           END_IF;
           //END_IF of IF #si_WDOG_RETRY < #si_WDOG_RETRY_NO 

         ELSE
           ;
           //keine Bedeutung 
         END_IF;
         //END_IF of IF #BUSY 

       END_IF;
       //END_IF of IF (NOT #BUSY AND #START AND NOT #sb_START_OLD) OR (#BUSY AND #sb_SEND)

     ELSE
       ;
       //Konfigurationsfehler: keine weitere Bearbeitung 

       #sb_CFG_ERR_1 := TRUE;

       //Auftrag ist nicht aktiv 

       #sb_BUSY := FALSE;

       //Auftrag fertig ruecksetzen 

       #sb_DONE := FALSE;
     END_IF;
     //END_IF of IF #LADDR <> 16#0000 

     //Flankenauswertung Startimpuls 

     #sb_START_OLD := #START;

     //CFG_ERR ausgeben 

     #CFG_ERR := #sb_CFG_ERR_1;

     //DB_ERR ausgeben 

     #DB_ERR := #sb_DB_ERR;

     // Initialisierung von Ausg㭧en
     #BUSY := #sb_BUSY;
     #DONE := #sb_DONE;
     #REQ_ERR := #sb_REQ_ERR;
END_FUNCTION_BLOCK

// ===== library: MasterCopy "DEV_FLT4" =====

FUNCTION_BLOCK "DEV_FLT4"   // FB39, SCL
TITLE = DEV_FLT4
{ S7_Optimized_Access := 'TRUE' }
AUTHOR : DRVDPS7
FAMILY : DRIVES
NAME : DEV_FLT4
VERSION : 5.0
// Read out fault buffer of a SINAMICS (CPU 1200)
   VAR_INPUT
      LADDR : Hw_Io;   // Logic base address of slot
      DS_NO : Word := 0;   // Number of data record
      AXIS : Byte;   // Axis addressing for multi-axis drives / Axis addressing
      START : Bool;   // Accept start impulse for request
   END_VAR
   VAR_OUTPUT
      BUSY : Bool;   // Request busy
      DONE : Bool := 1;   // Request completed without error
      REQ_ERR : Bool;   // Request completed with error
      WDOG_ERR : Bool;   // Watchdog error, no plausible response data exist
      SFB_ERR : Bool;   // SFB 53 WRREC / SFB 52 RDREC signals error
      CFG_ERR : Bool;   // Slave incorrectly configured or not at all
      ERR_NO1 : Word;   // Number fault 1 of fault event
      ERR_VAL1 : DWord;   // Fault value for fault number of fault 1
      ERR_NO2 : Word;   // Number fault 2 of fault event
      ERR_VAL2 : DWord;   // Fault value for fault number of fault 2
      ERR_NO3 : Word;   // Number fault 3 of fault event
      ERR_VAL3 : DWord;   // Fault value for fault number of fault 3
      ERR_NO4 : Word;   // Number fault 4 of fault event
      ERR_VAL4 : DWord;   // Fault value for fault number of fault 4
      ERR_NO5 : Word;   // Number fault 5 of fault event
      ERR_VAL5 : DWord;   // Fault value for fault number of fault 5
      ERR_NO6 : Word;   // Number fault 6 of fault event
      ERR_VAL6 : DWord;   // Fault value for fault number of fault 6
      ERR_NO7 : Word;   // Number fault 7 of fault event
      ERR_VAL7 : DWord;   // Fault value for fault number of fault 7
      ERR_NO8 : Word;   // Number fault 8 of fault event
      ERR_VAL8 : DWord;   // Fault value for fault number of fault 8 statische Variablen
   END_VAR
   VAR
      SFB53_RET_VAL : Int;   // Return value of SFB 53 WRREC
      SFB52_RET_VAL : Int;   // Return value of SFB 52 RDREC
      WDOG_RETRY_NO : Byte := BYTE#16#05;   // Number of request retries, when no plausible response data exists
      NODATA_RETRY_NO : Byte := BYTE#16#05;   // Number of request retries, when no response data exist
      NODATA_CYCLE_NO : Int := 2500;   // Number of cycles when no response data exist, before request retry
      sx_SEND_FA : Struct   // send buffer
         sy_AR : Byte;   // Auftragsreferenz
         sy_AKE : Byte := BYTE#16#01;   // Auftragskennung: 16#01 (Parameter anfordern )
         sy_A_NO : Byte := BYTE#16#00;   // Achsnummer
         sy_ANZ_PARA : Byte := BYTE#16#02;   // Anzahl Parameter: 16#02
         sy_ATTRIB1 : Byte := BYTE#16#10;   // Attribut: 16#10 (Wert)
         sy_ANZ_ELEM1 : Byte := BYTE#16#08;   // Anzahl Arrayelemente: 16#08
         si_PARA_NO1 : Int := 947;   // Parameternummer: 947 (Stoernummer)
         si_SUB_IND1 : Int := 0;   // Subindex: 0 (adressiert erstes Arrayelement auf das zugegriffen wird)
         sy_ATTRIB2 : Byte := BYTE#16#10;   // Attribut: 16#10 (Wert)
         sy_ANZ_ELEM2 : Byte := BYTE#16#08;   // Anzahl Arrayelemente: 16#08
         si_PARA_NO2 : Int := 949;   // Parameternummer: 949 (Stoerwert)
         si_SUB_IND2 : Int := 0;   // Subindex: 0 (adressiert erstes Arrayelement auf das zugegriffen wird)
      END_STRUCT;
      sx_RECV_FA : Struct   // receive buffer
         sy_AR : Byte;   // gespiegelte Auftragsreferenze
         sy_AKE : Byte;   // Antwortkennung
         sy_A_NO : Byte;   // Achsnummer
         sy_ANZ_PARA : Byte;   // Anzahl Parameter
         sy_FORMAT1 : Byte;   // Format
         sy_ANZ_VAL1 : Byte;   // Anzahl Werte
         sw_FAULT_NO1 : Word;   // Stoernummer 1
         sw_FAULT_NO2 : Word;   // Stoernummer 2
         sw_FAULT_NO3 : Word;   // Stoernummer 3
         sw_FAULT_NO4 : Word;   // Stoernummer 4
         sw_FAULT_NO5 : Word;   // Stoernummer 5
         sw_FAULT_NO6 : Word;   // Stoernummer 6
         sw_FAULT_NO7 : Word;   // Stoernummer 7
         sw_FAULT_NO8 : Word;   // Stoernummer 8
         sy_FORMAT2 : Byte;   // Format
         sy_ANZ_VAL2 : Byte;   // Anzahl Werte
         sd_FAULT_VAL1 : DWord;   // Stoerwert 1
         sd_FAULT_VAL2 : DWord;   // Stoerwert 2
         sd_FAULT_VAL3 : DWord;   // Stoerwert 3
         sd_FAULT_VAL4 : DWord;   // Stoerwert 4
         sd_FAULT_VAL5 : DWord;   // Stoerwert 5
         sd_FAULT_VAL6 : DWord;   // Stoerwert 6
         sd_FAULT_VAL7 : DWord;   // Stoerwert 7
         sd_FAULT_VAL8 : DWord;   // Stoerwert 8
      END_STRUCT;
      WDOG_RETRY : Byte;   // Counter for request retry for Watchdog monitoring
      NODATA_RETRY : Byte;   // Counter for request retry, if no response data exist
      NODATA_CYCLE : Int;   // Cycle counter, if no reponse data exist
      SEND_AC : Bool;   // Transmission active or request repetition for acyclic Communication
      START_AC : Bool;   // Start pulse for acyclic Communication
      BUSY_AC : Bool;   // Request busy for acyclic Communication
      READY_AC : Bool;   // Request completed without error for Acyclic communication
      SEND : Bool;   // send next request
      sb_DONE_AC : Bool;   // Stoerspeicher auslesen beendet
      sb_BUSY : Bool;   // Request busy
      sb_REQ_ERR : Bool;   // Request completed with error
      sb_WDOG_ERR : Bool;   // Watchdog error, no plausible response data exist
      sb_SFB_ERR : Bool;   // SFB 53 WRREC / SFB 52 RDREC signals error
      sb_CFG_ERR : Bool;   // Slave incorrectly configured or not at all
      si_AUF_REF : Int;   // Auftragsreferenz
      HM_RET_VAL : Int;   // Return value of SFB
      sb_START_OLD : Bool := 0;   // Start flag
      WRREC_1 : WRREC;   // Multiinstance of WRREC (SFB53)
      RDREC_1 : RDREC;   // Multiinstance of RDREC (SFB52) temporaere Variablen
   END_VAR
   VAR_TEMP
      pd_STATUS : DWord;   // STATUS der SFB's
      w_p_no : Word;   // Zwischenspeicher fuer Parameter-Nummer
      i_index : Int;   // Hilfsmerker fuer Index
      pi_LEN_RDREC : UInt;   // Tatsaechliche Laenge der empfangenen Daten
      pi_SFB_INDEX : Int;   // Index bei SFB52/53 Aufruf
      y_page_sel : Byte;   // Hilfsmerker PARA PAGE SELECT Funktion
      b_pind : Bool;   // Hilfsmerker Parameter-Index Sendefach Empfangsfach gleich
      b_busy : Bool;   // SFB 53 WRREC / SFB 52 RDREC sind beschaeftigt
      pb_DONE_WRREC : Bool;   // WRREC fertig
      pb_DONE_RDREC : Bool;   // RDREC fertig
      pb_ERR_WRREC : Bool;   // WRREC Fehler
      pb_ERR_RDREC : Bool;   // RDREC Fehler
   END_VAR
BEGIN
     //=============================================================================
     //SIEMENS AG
     //(c)Copyright 2017 All Rights Reserved
     //-----------------------------------------------------------------------------
     // Library: DriveLib
     // Tested with: S7-1200 CPU 1212C DC/DC/DC V4.1
     // Engineering: TIA Portal V14
     // Restrictions: -
     // Requirements: S7-1200
     // Functionality: The block reads out the last fault stored in the fault memory of the drive.
     //=============================================================================

     //Stoerungen lesen: Auftrag anstossen 

     //Startimpuls vorhanden und kein Auftrag aktiv 

     IF #START AND NOT #sb_BUSY AND NOT #sb_START_OLD
     THEN
       //Fehler / Ausgaenge abloeschen 

       #DONE := FALSE;
       #sb_REQ_ERR := FALSE;
       #sb_SFB_ERR := FALSE;
       #sb_CFG_ERR := FALSE;

       #sb_DONE_AC := FALSE;
     END_IF;
     //END_IF of IF #START AND NOT #BUSY AND NOT #sb_START_OLD

     //Startimpuls vorhanden oder Anforderung naechsten Auftrag zu senden vorhanden 

     IF #START AND NOT #sb_START_OLD OR #SEND
     THEN
       IF (#si_AUF_REF > 254) OR (#si_AUF_REF <= 0)
       THEN
         #si_AUF_REF := 1;
       ELSE
         ;
         #si_AUF_REF := #si_AUF_REF + 1;
       END_IF;
       //END_IF of IF (#si_AUF_REF > 254) OR (#si_AUF_REF <= 0)
       //Startimpuls fuer azyklischen Kommunikation setzen 

       #START_AC := TRUE;

       //Stoerungen auslesen ist aktiv 

       #sb_BUSY := TRUE;

       //Anforderung naechsten Auftrag senden ruecksetzen 

       #SEND := FALSE;
     ELSE
       ;
       //Startimpuls fuer azyklischen Kommunikation ruecksetzen 

       #START_AC := FALSE;
     END_IF;
     //END_IF of IF #START AND NOT #sb_START_OLD OR #SEND

     //Flankenauswertung Startimpuls 

     #sb_START_OLD := #START;

     //Ãœberpruefung, welcher Datensatz verwendet werden soll 

     #pi_SFB_INDEX := WORD_TO_INT(#DS_NO);

     IF #pi_SFB_INDEX = 0
     THEN
       #pi_SFB_INDEX := 47;
     ELSE
       ;
       ;    // not used
     END_IF;
     //END_IF of IF #pi_SFB_INDEX = 0

     //PDAT_AC2: Azyklische Kommunikation 

     //Hilfsmerker ruecksetzen 

     //Hilfsmerker ruecksetzen 

     #b_pind := FALSE;
     #y_page_sel := 16#00;
     #w_p_no := 16#0000;
     #i_index := 0;

     //Konfigurationsdaten pruefen: Slot = PKW-Slot und Logische Basisadresse <> 0 

     IF (#LADDR <> 16#0000)
     THEN
       //Konfiguration o.k. 

       #sb_CFG_ERR := FALSE;

       //Auftrag laeuft 

       IF #BUSY_AC
       THEN
         //Anzahl Zyklen, wenn keine Antwortdaten vorhanden, noch nicht abgelaufen  

         IF #NODATA_CYCLE < #NODATA_CYCLE_NO
         THEN
           //Anzahl Zyklen erhoehen 

           #NODATA_CYCLE := #NODATA_CYCLE + 1;
         ELSE
           ;
           //Fehler vorhanden: Return-Wert der SFBs < 0 

           IF #HM_RET_VAL < 0
           THEN
             //Keine Antwortdaten vorhanden oder temporaerer Fehler? 

             //Anzahl Auftragswiederholungen, wenn keine Antwortdaten vorhanden, noch nicht abgelaufen 

             IF #NODATA_RETRY < #NODATA_RETRY_NO
             THEN
               //Anzahl Auftragswiederholungen, wenn keine Antwortdaten vorhanden, erhoehen 

               #NODATA_RETRY := #NODATA_RETRY + 1;

               //Anzahl Zyklen initialisieren 

               #NODATA_CYCLE := 0;
             ELSE
               ;
               //SFB-Fehler 

               #sb_SFB_ERR := TRUE;

               IF #SEND_AC
               THEN
                 //Datensatz schreiben:                                                   
                 //Keine Antwortdaten vorhanden oder temporaerer Fehler, RET_VAL uebergeben 

                 #SFB53_RET_VAL := #HM_RET_VAL;
               ELSE
                 ;
                 //Datensatz lesen:                                                       
                 //Keine Antwortdaten vorhanden oder temporaerer Fehler, RET_VAL uebergeben 

                 #SFB52_RET_VAL := #HM_RET_VAL;
               END_IF;
               //END_IF of IF 
               //Auftragswiederholung ruecksetzen 

               #SEND_AC := FALSE;

               //Auftrag nicht aktiv 

               #BUSY_AC := FALSE;
             END_IF;
             //END_IF of IF #NODATA_RETRY < #NODATA_RETRY_NO
           END_IF;
           //END_IF of IF #HM_RET_VAL < 0
         END_IF;
         //END_IF of IF #NODATA_CYCLE < #NODATA_CYCLE_NO
       ELSE
         ;
         //Anzahl Zyklen und Anzahl Auftragswiederholungen initialisieren 

         #NODATA_CYCLE := 0;
         #NODATA_RETRY := 16#00;
         #WDOG_RETRY := 16#00;
       END_IF;
       //END_IF of IF #BUSY_AC
       //Auftrag nicht aktiv und Startimpuls vorhanden oder Senden aktiv oder Auftragswiederholung? 

       IF (NOT #BUSY_AC AND #START_AC) OR (#BUSY_AC AND #SEND_AC)
       THEN
         //Auftrag senden 

         //Fehler / Ausgaenge / Hilfsmerker ruecksetzen 

         //Startimpuls vorhanden und kein Senden bereits aktiv bzw. Auftragswiederholung? 

         IF (#START_AC = TRUE) AND (#SEND_AC = FALSE)
         THEN
           //Fehler / Ausgaenge / Hilfsmerker ruecksetzen 

           #READY_AC := FALSE;
           #sb_REQ_ERR := FALSE;
           #sb_WDOG_ERR := FALSE;
           #sb_SFB_ERR := FALSE;
           #SFB53_RET_VAL := 0;
           #SFB52_RET_VAL := 0;
         ELSE
           ;
         END_IF;
         //END_IF of IF (#START_AC = TRUE) AND (#SEND_AC = FALSE)
         #sx_SEND_FA.sy_AR := INT_TO_BYTE(#si_AUF_REF);                  // Auftragsreferenz
         #sx_SEND_FA.sy_AKE := 16#1;                                      // Auftragskennung: 16#01 (Parameter anfordern )
         #sx_SEND_FA.sy_A_NO := #AXIS;                                    // Achsnummer
         #sx_SEND_FA.sy_ANZ_PARA := 16#2;                                 // Anzahl Parameter: 16#02
         #sx_SEND_FA.sy_ATTRIB1 := 16#10;                                 // Attribut: 16#10 (Wert)
         #sx_SEND_FA.sy_ANZ_ELEM1 := 16#8;                                // Anzahl Arrayelemente: 16#08
         #sx_SEND_FA.si_PARA_NO1 := 947;                                  // Parameternummer: 947 (Stoernummer)
         #sx_SEND_FA.si_SUB_IND1 := 0;                                    // Subindex: 0 (adressiert erstes Arrayelement auf das zugegriffen wird)
         #sx_SEND_FA.sy_ATTRIB2 := 16#10;                                 // Attribut: 16#10 (Wert)
         #sx_SEND_FA.sy_ANZ_ELEM2 := 16#8;                                // Anzahl Arrayelemente: 16#08
         #sx_SEND_FA.si_PARA_NO2 := 949;                                  // Parameternummer: 949 (Stoerwert)
         #sx_SEND_FA.si_SUB_IND2 := 0;                                    // Subindex: 0 (adressiert erstes Arrayelement auf das zugegriffen wird)

         //Datenuebertragung: Auftrag senden (SFB53) 

         #WRREC_1(REQ := TRUE,
                  ID := #LADDR,
                  INDEX := #pi_SFB_INDEX,
                  LEN := 16,
                  RECORD := #sx_SEND_FA);
         #pb_DONE_WRREC := #WRREC_1.DONE;
         #b_busy := #WRREC_1.BUSY;
         #pb_ERR_WRREC := #WRREC_1.ERROR;
         #pd_STATUS := #WRREC_1.STATUS AND 16#FFFF00;
         #pd_STATUS := SHR(IN := #pd_STATUS, N := 8);

         #HM_RET_VAL := DWORD_TO_INT(#pd_STATUS);

         //Datenuebertragung beendet? 

         IF #b_busy = FALSE
         THEN
           //SFB-Fehler vorhanden? 

           IF #HM_RET_VAL < 0
           THEN
             //Temporaerer Fehler: RET_VAL <> 80A7, 80B5, 80C0, 80C1, 80C2, 80C3 oder 80C4 

             IF (#HM_RET_VAL <> -32601) AND (#HM_RET_VAL <> -32587) AND ((#HM_RET_VAL < -32576) OR (#HM_RET_VAL > -32572))
             THEN
               //SFB-Fehler 

               #sb_SFB_ERR := TRUE;

               //RET_VAL speichern 

               #SFB53_RET_VAL := #HM_RET_VAL;

               //Senden aktiv / Auftragswiederholung ruecksetzen 

               #SEND_AC := FALSE;

               //Auftrag ist nicht aktiv 

               #BUSY_AC := FALSE;
             ELSE
               ;
               //Auftrag ist aktiv 

               #BUSY_AC := TRUE;

               //Senden aktiv setzen, Auftrag wird noch einmal geschrieben. 

               #SEND_AC := TRUE;
             END_IF;
             //END_IF of IF (#HM_RET_VAL <> -32601) AND (#HM_RET_VAL <> -32587) AND ((#HM_RET_VAL < -32576) OR (#HM_RET_VAL > -32572))
           ELSE
             ;
             //Auftrag ist aktiv 

             #BUSY_AC := TRUE;

             //Senden aktiv / Auftragswiederholung ruecksetzen 

             #SEND_AC := FALSE;
           END_IF;
           //END_IF of IF #HM_RET_VAL < 0
         ELSE
           ;
           //Auftrag ist aktiv 

           #BUSY_AC := TRUE;

           //Senden aktiv setzen 

           #SEND_AC := TRUE;
         END_IF;
         //END_IF of IF #b_busy = FALSE
       ELSE
         ;
         //Auftrag laeuft 

         IF #BUSY_AC
         THEN
           //Anzahl Auftragswiederholungen fuer Watchdog noch nicht abgelaufen 

           IF #WDOG_RETRY < #WDOG_RETRY_NO
           THEN
             //Auftrag empfangen 

             //Datenuebertragung: Auftrag empfangen 

             #RDREC_1(REQ := TRUE,
                      ID := #LADDR,
                      INDEX := #pi_SFB_INDEX,
                      MLEN := 56,
                      RECORD := #sx_RECV_FA);

             #pb_DONE_RDREC := #RDREC_1.VALID;
             #b_busy := #RDREC_1.BUSY;
             #pb_ERR_RDREC := #RDREC_1.ERROR;
             #pd_STATUS := #RDREC_1.STATUS AND 16#FFFF00;
             #pi_LEN_RDREC := #RDREC_1.LEN;

             #pd_STATUS := SHR(IN := #pd_STATUS, N := 8);
             #HM_RET_VAL := DWORD_TO_INT(#pd_STATUS);

             //Datenuebertragung beendet? 

             IF #b_busy = FALSE
             THEN
               //SFB-Fehler vorhanden? 

               IF #HM_RET_VAL < 0
               THEN
                 //Temporaerer Fehler: RET_VAL <> 80A7, 80B5, 80C0, 80C1, 80C2, 80C3 oder 80C4 

                 IF (#HM_RET_VAL <> -32601) AND (#HM_RET_VAL <> -32587) AND ((#HM_RET_VAL < -32576) OR (#HM_RET_VAL > -32572))
                 THEN
                   //SFB-Fehler 

                   #sb_SFB_ERR := TRUE;

                   //Auftrag ist nicht aktiv 

                   #BUSY_AC := FALSE;

                   //RET_VAL speichern 

                   #SFB52_RET_VAL := #HM_RET_VAL;

                   //Ausgaenge abloeschen 

                   #ERR_NO1 := 0;
                   #ERR_VAL1 := 0;
                   #ERR_NO2 := 0;
                   #ERR_VAL2 := 0;
                   #ERR_NO3 := 0;
                   #ERR_VAL3 := 0;
                   #ERR_NO4 := 0;
                   #ERR_VAL4 := 0;
                   #ERR_NO5 := 0;
                   #ERR_VAL5 := 0;
                   #ERR_NO6 := 0;
                   #ERR_VAL6 := 0;
                   #ERR_NO7 := 0;
                   #ERR_VAL7 := 0;
                   #ERR_NO8 := 0;
                   #ERR_VAL8 := 0;
                 ELSE
                   ;
                   //keine Bedeutung 
                 END_IF;
                 //END_IF of IF (#HM_RET_VAL <> -32601) AND (#HM_RET_VAL <> -32587) AND ((#HM_RET_VAL < -32576) OR (#HM_RET_VAL > -32572))

               ELSE
                 ;
                 //Antwortdaten auswerten 

                 IF #sx_SEND_FA.sy_AR = #sx_RECV_FA.sy_AR
                 THEN
                   IF #sx_RECV_FA.sy_AKE = 16#81 OR #sx_RECV_FA.sy_AKE = 16#82
                   THEN
                     #sb_REQ_ERR := TRUE;

                     #sb_DONE_AC := FALSE;
                   ELSE
                     ;
                     #sb_REQ_ERR := FALSE;

                     #sb_DONE_AC := TRUE;
                   END_IF;
                   //END_IF of IF #sx_RECV_FA.sy_AKE = 16#81 OR #sx_RECV_FA.sy_AKE = 16#82

                 ELSE
                   ;
                   //keine Bedeutung 
                 END_IF;
                 //END_IF of IF #sx_SEND_FA.sy_AR = #sx_RECV_FA.sy_AR

                 //Auftrag fertig ohne Fehler 

                 IF #sb_DONE_AC
                 THEN
                   //Stoernummer 

                   #ERR_NO1 := #sx_RECV_FA.sw_FAULT_NO1;
                   #ERR_NO2 := #sx_RECV_FA.sw_FAULT_NO2;
                   #ERR_NO3 := #sx_RECV_FA.sw_FAULT_NO3;
                   #ERR_NO4 := #sx_RECV_FA.sw_FAULT_NO4;
                   #ERR_NO5 := #sx_RECV_FA.sw_FAULT_NO5;
                   #ERR_NO6 := #sx_RECV_FA.sw_FAULT_NO6;
                   #ERR_NO7 := #sx_RECV_FA.sw_FAULT_NO7;
                   #ERR_NO8 := #sx_RECV_FA.sw_FAULT_NO8;

                   //Stoerwert 

                   #ERR_VAL1 := #sx_RECV_FA.sd_FAULT_VAL1;
                   #ERR_VAL2 := #sx_RECV_FA.sd_FAULT_VAL2;
                   #ERR_VAL3 := #sx_RECV_FA.sd_FAULT_VAL3;
                   #ERR_VAL4 := #sx_RECV_FA.sd_FAULT_VAL4;
                   #ERR_VAL5 := #sx_RECV_FA.sd_FAULT_VAL5;
                   #ERR_VAL6 := #sx_RECV_FA.sd_FAULT_VAL6;
                   #ERR_VAL7 := #sx_RECV_FA.sd_FAULT_VAL7;
                   #ERR_VAL8 := #sx_RECV_FA.sd_FAULT_VAL8;

                   //Auftrag ist nicht aktiv 

                   #BUSY_AC := FALSE;

                   //Auftrag fertig mit Fehler 

                 ELSIF #sb_REQ_ERR
                 THEN
                   //Ausgaenge abloeschen 

                   #ERR_NO1 := 0;
                   #ERR_VAL1 := 0;
                   #ERR_NO2 := 0;
                   #ERR_VAL2 := 0;
                   #ERR_NO3 := 0;
                   #ERR_VAL3 := 0;
                   #ERR_NO4 := 0;
                   #ERR_VAL4 := 0;
                   #ERR_NO5 := 0;
                   #ERR_VAL5 := 0;
                   #ERR_NO6 := 0;
                   #ERR_VAL6 := 0;
                   #ERR_NO7 := 0;
                   #ERR_VAL7 := 0;
                   #ERR_NO8 := 0;
                   #ERR_VAL8 := 0;

                   //Auftrag ist nicht aktiv 

                   #BUSY_AC := FALSE;

                 ELSE
                   //Anzahl Auftragswiederholungen, wenn keine plausiblen Antwortdaten vorhanden, erhoehen 

                   #WDOG_RETRY := #WDOG_RETRY + 1;

                   //Anzahl Zyklen initialisieren 

                   #NODATA_CYCLE := 0;

                   //Auftragswiederholung anstossen 

                   #SEND_AC := TRUE;
                 END_IF;
                 //END_IF of IF #sb_DONE_AC

               END_IF;
               //END_IF of IF #HM_RET_VAL < 0

             END_IF;
             //END_IF of IF #b_busy = FALSE

           ELSE
             ;
             //Watchdog-     
             //Fehler melden 

             #sb_WDOG_ERR := TRUE;

             //Auftrag ist nicht aktiv 

             #BUSY_AC := FALSE;
           END_IF;
           //END_IF of IF #WDOG_RETRY < #WDOG_RETRY_NO

         ELSE
           ;
           //Nein: Keine Bearbeitung 
         END_IF;
         //END_IF of IF #BUSY_AC
       END_IF;
       //END_IF of IF (NOT #BUSY_AC AND #START_AC) OR (#BUSY_AC AND #SEND_AC)
     ELSE
       ;
       //Konfigurationsfehler: Keine weitere Bearbeitung 

       #sb_CFG_ERR := TRUE;

       //Auftrag ist nicht aktiv 

       #BUSY_AC := FALSE;

       //Auftrag fertig ruecksetzen 

       #READY_AC := FALSE;
     END_IF;
     //END_IF of IF (#LADDR <> 16#0000)

     //Stoerungen auslesen: Antwort auswerten 

     //Stoerungen auslesen laeuft 

     IF #sb_BUSY
     THEN
       //Auftrag fertig 

       IF #sb_DONE_AC
       THEN
         //Auftrag fertig ohne Fehler 

         #DONE := TRUE;

         //Auftrag ist nicht aktiv 

         #sb_BUSY := FALSE;
       ELSE
         ;
         //Fehler aufgetreten waehrend der Kommunikation 

         IF #sb_REQ_ERR OR #sb_WDOG_ERR OR #sb_SFB_ERR OR #sb_CFG_ERR
         THEN
           //Auftrag ist nicht aktiv 

           #sb_BUSY := FALSE;

           //Auftrag ist nicht fertig 

           #DONE := FALSE;
         END_IF;
         //END_IF of IF #REQ_ERR OR #WDOG_ERR OR #SFB_ERR OR #CFG_ERR
       END_IF;
       //END_IF of IF #sb_DONE_AC
     END_IF;
     //END_IF of IF #BUSY

     // Initialisierung von Ausg㭧en
     #BUSY := #sb_BUSY;
     #REQ_ERR := #sb_REQ_ERR;
     #WDOG_ERR := #sb_WDOG_ERR;
     #SFB_ERR := #sb_SFB_ERR;
     #CFG_ERR := #sb_CFG_ERR;
END_FUNCTION_BLOCK

// ===== library: MasterCopy "SLOT_UDT" =====

TYPE "SLOT_UDT"
   STRUCT
      LADDR : HW_IO;   // I/O base address of slot
      SLOT_ID : Byte;   // Slot type ID
      PCD_ADDR : Byte;   // Process data address
      LENGTH : Byte;   // Slot data length
      CONSIST : Bool;   // Consistency condition
   END_STRUCT;
END_TYPE

// ===== library: MasterCopy "DEV_FLT4" =====

FUNCTION_BLOCK "DEV_FLT4"   // FB39, SCL
TITLE = DEV_FLT4
{ S7_Optimized_Access := 'FALSE' }
AUTHOR : DRVDPS7
FAMILY : DRIVES
NAME : DEV_FLT4
VERSION : 5.0
// Read out fault buffer of a SINAMICS (CPU 1500)
   VAR_INPUT
      LADDR : HW_IO;   // Logic base address of slot
      DS_NO : Word := 0;   // Number of data record
      AXIS : Byte;   // Axis addressing for multi-axis drives / Axis addressing
      START : Bool;   // Accept start impulse for request
   END_VAR
   VAR_OUTPUT
      BUSY : Bool;   // Request busy
      DONE : Bool := 1;   // Request completed without error
      REQ_ERR : Bool;   // Request completed with error
      WDOG_ERR : Bool;   // Watchdog error, no plausible response data exist
      SFB_ERR : Bool;   // SFB 53 WRREC / SFB 52 RDREC signals error
      CFG_ERR : Bool;   // Slave incorrectly configured or not at all
      ERR_NO1 : Word;   // Number fault 1 of fault event
      ERR_VAL1 : DWord;   // Fault value for fault number of fault 1
      ERR_NO2 : Word;   // Number fault 2 of fault event
      ERR_VAL2 : DWord;   // Fault value for fault number of fault 2
      ERR_NO3 : Word;   // Number fault 3 of fault event
      ERR_VAL3 : DWord;   // Fault value for fault number of fault 3
      ERR_NO4 : Word;   // Number fault 4 of fault event
      ERR_VAL4 : DWord;   // Fault value for fault number of fault 4
      ERR_NO5 : Word;   // Number fault 5 of fault event
      ERR_VAL5 : DWord;   // Fault value for fault number of fault 5
      ERR_NO6 : Word;   // Number fault 6 of fault event
      ERR_VAL6 : DWord;   // Fault value for fault number of fault 6
      ERR_NO7 : Word;   // Number fault 7 of fault event
      ERR_VAL7 : DWord;   // Fault value for fault number of fault 7
      ERR_NO8 : Word;   // Number fault 8 of fault event
      ERR_VAL8 : DWord;   // Fault value for fault number of fault 8 statische Variablen
   END_VAR
   VAR
      SFB53_RET_VAL : Int;   // Return value of SFB 53 WRREC
      SFB52_RET_VAL : Int;   // Return value of SFB 52 RDREC
      WDOG_RETRY_NO : Byte := BYTE#16#05;   // Number of request retries, when no plausible response data exists
      NODATA_RETRY_NO : Byte := BYTE#16#05;   // Number of request retries, when no response data exist
      NODATA_CYCLE_NO : Int := 2500;   // Number of cycles when no response data exist, before request retry Variablen fuer Stoerspeicher auslesen
      sx_SEND_FA : Struct
         sy_AR : Byte;   // Auftragsreferenz
         sy_AKE : Byte := BYTE#16#01;   // Auftragskennung: 16#01 (Parameter anfordern )
         sy_A_NO : Byte := BYTE#16#00;   // Achsnummer
         sy_ANZ_PARA : Byte := BYTE#16#02;   // Anzahl Parameter: 16#02
         sy_ATTRIB1 : Byte := BYTE#16#10;   // Attribut: 16#10 (Wert)
         sy_ANZ_ELEM1 : Byte := BYTE#16#08;   // Anzahl Arrayelemente: 16#08
         si_PARA_NO1 : Int := 947;   // Parameternummer: 947 (Stoernummer)
         si_SUB_IND1 : Int := 0;   // Subindex: 0 (adressiert erstes Arrayelement auf das zugegriffen wird)
         sy_ATTRIB2 : Byte := BYTE#16#10;   // Attribut: 16#10 (Wert)
         sy_ANZ_ELEM2 : Byte := BYTE#16#08;   // Anzahl Arrayelemente: 16#08
         si_PARA_NO2 : Int := 949;   // Parameternummer: 949 (Stoerwert)
         si_SUB_IND2 : Int := 0;   // Subindex: 0 (adressiert erstes Arrayelement auf das zugegriffen wird)
      END_STRUCT;
      sx_RECV_FA : Struct
         sy_AR : Byte;   // gespiegelte Auftragsreferenze
         sy_AKE : Byte;   // Antwortkennung
         sy_A_NO : Byte;   // Achsnummer
         sy_ANZ_PARA : Byte;   // Anzahl Parameter
         sy_FORMAT1 : Byte;   // Format
         sy_ANZ_VAL1 : Byte;   // Anzahl Werte
         sw_FAULT_NO1 : Word;   // Stoernummer 1
         sw_FAULT_NO2 : Word;   // Stoernummer 2
         sw_FAULT_NO3 : Word;   // Stoernummer 3
         sw_FAULT_NO4 : Word;   // Stoernummer 4
         sw_FAULT_NO5 : Word;   // Stoernummer 5
         sw_FAULT_NO6 : Word;   // Stoernummer 6
         sw_FAULT_NO7 : Word;   // Stoernummer 7
         sw_FAULT_NO8 : Word;   // Stoernummer 8
         sy_FORMAT2 : Byte;   // Format
         sy_ANZ_VAL2 : Byte;   // Anzahl Werte
         sd_FAULT_VAL1 : DWord;   // Stoerwert 1
         sd_FAULT_VAL2 : DWord;   // Stoerwert 2
         sd_FAULT_VAL3 : DWord;   // Stoerwert 3
         sd_FAULT_VAL4 : DWord;   // Stoerwert 4
         sd_FAULT_VAL5 : DWord;   // Stoerwert 5
         sd_FAULT_VAL6 : DWord;   // Stoerwert 6
         sd_FAULT_VAL7 : DWord;   // Stoerwert 7
         sd_FAULT_VAL8 : DWord;   // Stoerwert 8
      END_STRUCT;
      WDOG_RETRY : Byte;   // Counter for request retry for Watchdog monitoring
      NODATA_RETRY : Byte;   // Counter for request retry, if no response data exist
      NODATA_CYCLE : Int;   // Cycle counter, if no reponse data exist
      SEND_AC : Bool;   // Transmission active or request repetition for acyclic Communication
      START_AC : Bool;   // Start pulse for acyclic Communication
      BUSY_AC : Bool;   // Request busy for acyclic Communication
      READY_AC : Bool;   // Request completed without error for Acyclic communication
      SEND : Bool;   // send next request
      sb_DONE_AC : Bool;   // Stoerspeicher auslesen beendet
      sb_BUSY : Bool;   // Request busy
      sb_REQ_ERR : Bool;   // REQ_ERR
      sb_WDOG_ERR : Bool;   // Watchdog error, no plausible response data exist
      sb_SFB_ERR : Bool;   // SFB 53 WRREC / SFB 52 RDREC signals error
      sb_CFG_ERR : Bool;   // Slave incorrectly configured or not at all
      si_AUF_REF : Int;   // Auftragsreferenz
      HM_RET_VAL : Int;   // Return value of SFB
      sb_START_OLD : Bool := 0;   // Start flag
      WRREC_1 : WRREC;   // Multiinstance of WRREC (SFB53)
      RDREC_1 : RDREC;   // Multiinstance of RDREC (SFB52) temporaere Variablen
   END_VAR
   VAR_TEMP
      pd_STATUS : DWord;   // STATUS der SFB's
      w_p_no : Word;   // Zwischenspeicher fuer Parameter-Nummer
      i_index : Int;   // Hilfsmerker fuer Index
      pi_LEN_RDREC : UInt;   // Tatsaechliche Laenge der empfangenen Daten
      pi_SFB_INDEX : Int;   // Index bei SFB52/53 Aufruf
      y_page_sel : Byte;   // Hilfsmerker PARA PAGE SELECT Funktion
      b_pind : Bool;   // Hilfsmerker Parameter-Index Sendefach Empfangsfach gleich
      b_busy : Bool;   // SFB 53 WRREC / SFB 52 RDREC sind beschaeftigt
      pb_DONE_WRREC : Bool;   // WRREC fertig
      pb_DONE_RDREC : Bool;   // RDREC fertig
      pb_ERR_WRREC : Bool;   // WRREC Fehler
      pb_ERR_RDREC : Bool;   // RDREC Fehler
   END_VAR
BEGIN
     //=============================================================================
     //SIEMENS AG
     //(c)Copyright 2017 All Rights Reserved
     //-----------------------------------------------------------------------------
     // Library: DriveLib
     // Tested with: S7-1516-3 PN/DP V1.8
     // Engineering: TIA Portal V14
     // Restrictions: -
     // Requirements: S7-1500
     // Functionality: The block reads out the last fault stored in the fault memory of the drive.
     //=============================================================================

     //Stoerungen lesen: Auftrag anstossen 

     //Startimpuls vorhanden und kein Auftrag aktiv 

     IF #START AND NOT #sb_BUSY AND NOT #sb_START_OLD
     THEN
       //Fehler / Ausgaenge abloeschen 

       #DONE := FALSE;
       #sb_REQ_ERR := FALSE;
       #sb_SFB_ERR := FALSE;
       #sb_CFG_ERR := FALSE;

       #sb_DONE_AC := FALSE;
     END_IF;
     //END_IF of IF #START AND NOT #BUSY AND NOT #sb_START_OLD

     //Startimpuls vorhanden oder Anforderung naechsten Auftrag zu senden vorhanden 

     IF #START AND NOT #sb_START_OLD OR #SEND
     THEN
       IF (#si_AUF_REF > 254) OR (#si_AUF_REF <= 0)
       THEN
         #si_AUF_REF := 1;
       ELSE
         ;
         #si_AUF_REF := #si_AUF_REF + 1;
       END_IF;
       //END_IF of IF (#si_AUF_REF > 254) OR (#si_AUF_REF <= 0)
       //Startimpuls fuer azyklischen Kommunikation setzen 

       #START_AC := TRUE;

       //Stoerungen auslesen ist aktiv 

       #sb_BUSY := TRUE;

       //Anforderung naechsten Auftrag senden ruecksetzen 

       #SEND := FALSE;
     ELSE
       ;
       //Startimpuls fuer azyklischen Kommunikation ruecksetzen 

       #START_AC := FALSE;
     END_IF;
     //END_IF of IF #START AND NOT #sb_START_OLD OR #SEND

     //Flankenauswertung Startimpuls 

     #sb_START_OLD := #START;

     //ÃƒÅ“berpruefung, welcher Datensatz verwendet werden soll 

     #pi_SFB_INDEX := WORD_TO_INT(#DS_NO);

     IF #pi_SFB_INDEX = 0
     THEN
       #pi_SFB_INDEX := 47;
     ELSE
       ;
       ;    // not used
     END_IF;
     //END_IF of IF #pi_SFB_INDEX = 0

     //PDAT_AC2: Azyklische Kommunikation 

     //Hilfsmerker ruecksetzen 

     //Hilfsmerker ruecksetzen 

     #b_pind := FALSE;
     #y_page_sel := 16#00;
     #w_p_no := 16#0000;
     #i_index := 0;

     //Konfigurationsdaten pruefen: Slot = PKW-Slot und Logische Basisadresse <> 0 

     IF (#LADDR <> 16#0000)
     THEN
       //Konfiguration o.k. 

       #sb_CFG_ERR := FALSE;

       //Auftrag laeuft 

       IF #BUSY_AC
       THEN
         //Anzahl Zyklen, wenn keine Antwortdaten vorhanden, noch nicht abgelaufen  

         IF #NODATA_CYCLE < #NODATA_CYCLE_NO
         THEN
           //Anzahl Zyklen erhoehen 

           #NODATA_CYCLE := #NODATA_CYCLE + 1;
         ELSE
           ;
           //Fehler vorhanden: Return-Wert der SFBs < 0 

           IF #HM_RET_VAL < 0
           THEN
             //Keine Antwortdaten vorhanden oder temporaerer Fehler? 

             //Anzahl Auftragswiederholungen, wenn keine Antwortdaten vorhanden, noch nicht abgelaufen 

             IF #NODATA_RETRY < #NODATA_RETRY_NO
             THEN
               //Anzahl Auftragswiederholungen, wenn keine Antwortdaten vorhanden, erhoehen 

               #NODATA_RETRY := #NODATA_RETRY + 1;

               //Anzahl Zyklen initialisieren 

               #NODATA_CYCLE := 0;
             ELSE
               ;
               //SFB-Fehler 

               #sb_SFB_ERR := TRUE;

               IF #SEND_AC
               THEN
                 //Datensatz schreiben:                                                   
                 //Keine Antwortdaten vorhanden oder temporaerer Fehler, RET_VAL uebergeben 

                 #SFB53_RET_VAL := #HM_RET_VAL;
               ELSE
                 ;
                 //Datensatz lesen:                                                       
                 //Keine Antwortdaten vorhanden oder temporaerer Fehler, RET_VAL uebergeben 

                 #SFB52_RET_VAL := #HM_RET_VAL;
               END_IF;
               //END_IF of IF 
               //Auftragswiederholung ruecksetzen 

               #SEND_AC := FALSE;

               //Auftrag nicht aktiv 

               #BUSY_AC := FALSE;
             END_IF;
             //END_IF of IF #NODATA_RETRY < #NODATA_RETRY_NO
           END_IF;
           //END_IF of IF #HM_RET_VAL < 0
         END_IF;
         //END_IF of IF #NODATA_CYCLE < #NODATA_CYCLE_NO
       ELSE
         ;
         //Anzahl Zyklen und Anzahl Auftragswiederholungen initialisieren 

         #NODATA_CYCLE := 0;
         #NODATA_RETRY := 16#00;
         #WDOG_RETRY := 16#00;
       END_IF;
       //END_IF of IF #BUSY_AC
       //Auftrag nicht aktiv und Startimpuls vorhanden oder Senden aktiv oder Auftragswiederholung? 

       IF (NOT #BUSY_AC AND #START_AC) OR (#BUSY_AC AND #SEND_AC)
       THEN
         //Auftrag senden 

         //Fehler / Ausgaenge / Hilfsmerker ruecksetzen 

         //Startimpuls vorhanden und kein Senden bereits aktiv bzw. Auftragswiederholung? 

         IF (#START_AC = TRUE) AND (#SEND_AC = FALSE)
         THEN
           //Fehler / Ausgaenge / Hilfsmerker ruecksetzen 

           #READY_AC := FALSE;
           #sb_REQ_ERR := FALSE;
           #sb_WDOG_ERR := FALSE;
           #sb_SFB_ERR := FALSE;
           #SFB53_RET_VAL := 0;
           #SFB52_RET_VAL := 0;
         ELSE
           ;
         END_IF;
         //END_IF of IF (#START_AC = TRUE) AND (#SEND_AC = FALSE)
         #sx_SEND_FA.sy_AR := INT_TO_BYTE(#si_AUF_REF);                  // Auftragsreferenz
         #sx_SEND_FA.sy_AKE := 16#1;                                      // Auftragskennung: 16#01 (Parameter anfordern )
         #sx_SEND_FA.sy_A_NO := #AXIS;                                    // Achsnummer
         #sx_SEND_FA.sy_ANZ_PARA := 16#2;                                 // Anzahl Parameter: 16#02
         #sx_SEND_FA.sy_ATTRIB1 := 16#10;                                 // Attribut: 16#10 (Wert)
         #sx_SEND_FA.sy_ANZ_ELEM1 := 16#8;                                // Anzahl Arrayelemente: 16#08
         #sx_SEND_FA.si_PARA_NO1 := 947;                                  // Parameternummer: 947 (Stoernummer)
         #sx_SEND_FA.si_SUB_IND1 := 0;                                    // Subindex: 0 (adressiert erstes Arrayelement auf das zugegriffen wird)
         #sx_SEND_FA.sy_ATTRIB2 := 16#10;                                 // Attribut: 16#10 (Wert)
         #sx_SEND_FA.sy_ANZ_ELEM2 := 16#8;                                // Anzahl Arrayelemente: 16#08
         #sx_SEND_FA.si_PARA_NO2 := 949;                                  // Parameternummer: 949 (Stoerwert)
         #sx_SEND_FA.si_SUB_IND2 := 0;                                    // Subindex: 0 (adressiert erstes Arrayelement auf das zugegriffen wird)

         //Datenuebertragung: Auftrag senden (SFB53) 

         #WRREC_1(REQ := TRUE,
                  ID := #LADDR,
                  INDEX := #pi_SFB_INDEX,
                  LEN := 16,
                  RECORD := #sx_SEND_FA);
         #pb_DONE_WRREC := #WRREC_1.DONE;
         #b_busy := #WRREC_1.BUSY;
         #pb_ERR_WRREC := #WRREC_1.ERROR;
         #pd_STATUS := #WRREC_1.STATUS AND 16#FFFF00;
         #pd_STATUS := SHR(IN := #pd_STATUS, N := 8);

         #HM_RET_VAL := DWORD_TO_INT(#pd_STATUS);

         //Datenuebertragung beendet? 

         IF #b_busy = FALSE
         THEN
           //SFB-Fehler vorhanden? 

           IF #HM_RET_VAL < 0
           THEN
             //Temporaerer Fehler: RET_VAL <> 80A7, 80B5, 80C0, 80C1, 80C2, 80C3 oder 80C4 

             IF (#HM_RET_VAL <> -32601) AND (#HM_RET_VAL <> -32587) AND ((#HM_RET_VAL < -32576) OR (#HM_RET_VAL > -32572))
             THEN
               //SFB-Fehler 

               #sb_SFB_ERR := TRUE;

               //RET_VAL speichern 

               #SFB53_RET_VAL := #HM_RET_VAL;

               //Senden aktiv / Auftragswiederholung ruecksetzen 

               #SEND_AC := FALSE;

               //Auftrag ist nicht aktiv 

               #BUSY_AC := FALSE;
             ELSE
               ;
               //Auftrag ist aktiv 

               #BUSY_AC := TRUE;

               //Senden aktiv setzen, Auftrag wird noch einmal geschrieben. 

               #SEND_AC := TRUE;
             END_IF;
             //END_IF of IF (#HM_RET_VAL <> -32601) AND (#HM_RET_VAL <> -32587) AND ((#HM_RET_VAL < -32576) OR (#HM_RET_VAL > -32572))
           ELSE
             ;
             //Auftrag ist aktiv 

             #BUSY_AC := TRUE;

             //Senden aktiv / Auftragswiederholung ruecksetzen 

             #SEND_AC := FALSE;
           END_IF;
           //END_IF of IF #HM_RET_VAL < 0
         ELSE
           ;
           //Auftrag ist aktiv 

           #BUSY_AC := TRUE;

           //Senden aktiv setzen 

           #SEND_AC := TRUE;
         END_IF;
         //END_IF of IF #b_busy = FALSE
       ELSE
         ;
         //Auftrag laeuft 

         IF #BUSY_AC
         THEN
           //Anzahl Auftragswiederholungen fuer Watchdog noch nicht abgelaufen 

           IF #WDOG_RETRY < #WDOG_RETRY_NO
           THEN
             //Auftrag empfangen 

             //Datenuebertragung: Auftrag empfangen 

             #RDREC_1(REQ := TRUE,
                      ID := #LADDR,
                      INDEX := #pi_SFB_INDEX,
                      MLEN := 56,
                      RECORD := #sx_RECV_FA);

             #pb_DONE_RDREC := #RDREC_1.VALID;
             #b_busy := #RDREC_1.BUSY;
             #pb_ERR_RDREC := #RDREC_1.ERROR;
             #pd_STATUS := #RDREC_1.STATUS AND 16#FFFF00;
             #pi_LEN_RDREC := #RDREC_1.LEN;

             #pd_STATUS := SHR(IN := #pd_STATUS, N := 8);
             #HM_RET_VAL := DWORD_TO_INT(#pd_STATUS);

             //Datenuebertragung beendet? 

             IF #b_busy = FALSE
             THEN
               //SFB-Fehler vorhanden? 

               IF #HM_RET_VAL < 0
               THEN
                 //Temporaerer Fehler: RET_VAL <> 80A7, 80B5, 80C0, 80C1, 80C2, 80C3 oder 80C4 

                 IF (#HM_RET_VAL <> -32601) AND (#HM_RET_VAL <> -32587) AND ((#HM_RET_VAL < -32576) OR (#HM_RET_VAL > -32572))
                 THEN
                   //SFB-Fehler 

                   #sb_SFB_ERR := TRUE;

                   //Auftrag ist nicht aktiv 

                   #BUSY_AC := FALSE;

                   //RET_VAL speichern 

                   #SFB52_RET_VAL := #HM_RET_VAL;

                   //Ausgaenge abloeschen 

                   #ERR_NO1 := 0;
                   #ERR_VAL1 := 0;
                   #ERR_NO2 := 0;
                   #ERR_VAL2 := 0;
                   #ERR_NO3 := 0;
                   #ERR_VAL3 := 0;
                   #ERR_NO4 := 0;
                   #ERR_VAL4 := 0;
                   #ERR_NO5 := 0;
                   #ERR_VAL5 := 0;
                   #ERR_NO6 := 0;
                   #ERR_VAL6 := 0;
                   #ERR_NO7 := 0;
                   #ERR_VAL7 := 0;
                   #ERR_NO8 := 0;
                   #ERR_VAL8 := 0;
                 ELSE
                   ;
                   //keine Bedeutung 
                 END_IF;
                 //END_IF of IF (#HM_RET_VAL <> -32601) AND (#HM_RET_VAL <> -32587) AND ((#HM_RET_VAL < -32576) OR (#HM_RET_VAL > -32572))

               ELSE
                 ;
                 //Antwortdaten auswerten 

                 IF #sx_SEND_FA.sy_AR = #sx_RECV_FA.sy_AR
                 THEN
                   IF #sx_RECV_FA.sy_AKE = 16#81 OR #sx_RECV_FA.sy_AKE = 16#82
                   THEN
                     #sb_REQ_ERR := TRUE;

                     #sb_DONE_AC := FALSE;
                   ELSE
                     ;
                     #sb_REQ_ERR := FALSE;

                     #sb_DONE_AC := TRUE;
                   END_IF;
                   //END_IF of IF #sx_RECV_FA.sy_AKE = 16#81 OR #sx_RECV_FA.sy_AKE = 16#82

                 ELSE
                   ;
                   //keine Bedeutung 
                 END_IF;
                 //END_IF of IF #sx_SEND_FA.sy_AR = #sx_RECV_FA.sy_AR

                 //Auftrag fertig ohne Fehler 

                 IF #sb_DONE_AC
                 THEN
                   //Stoernummer 

                   #ERR_NO1 := #sx_RECV_FA.sw_FAULT_NO1;
                   #ERR_NO2 := #sx_RECV_FA.sw_FAULT_NO2;
                   #ERR_NO3 := #sx_RECV_FA.sw_FAULT_NO3;
                   #ERR_NO4 := #sx_RECV_FA.sw_FAULT_NO4;
                   #ERR_NO5 := #sx_RECV_FA.sw_FAULT_NO5;
                   #ERR_NO6 := #sx_RECV_FA.sw_FAULT_NO6;
                   #ERR_NO7 := #sx_RECV_FA.sw_FAULT_NO7;
                   #ERR_NO8 := #sx_RECV_FA.sw_FAULT_NO8;

                   //Stoerwert 

                   #ERR_VAL1 := #sx_RECV_FA.sd_FAULT_VAL1;
                   #ERR_VAL2 := #sx_RECV_FA.sd_FAULT_VAL2;
                   #ERR_VAL3 := #sx_RECV_FA.sd_FAULT_VAL3;
                   #ERR_VAL4 := #sx_RECV_FA.sd_FAULT_VAL4;
                   #ERR_VAL5 := #sx_RECV_FA.sd_FAULT_VAL5;
                   #ERR_VAL6 := #sx_RECV_FA.sd_FAULT_VAL6;
                   #ERR_VAL7 := #sx_RECV_FA.sd_FAULT_VAL7;
                   #ERR_VAL8 := #sx_RECV_FA.sd_FAULT_VAL8;

                   //Auftrag ist nicht aktiv 

                   #BUSY_AC := FALSE;

                   //Auftrag fertig mit Fehler 

                 ELSIF #sb_REQ_ERR
                 THEN
                   //Ausgaenge abloeschen 

                   #ERR_NO1 := 0;
                   #ERR_VAL1 := 0;
                   #ERR_NO2 := 0;
                   #ERR_VAL2 := 0;
                   #ERR_NO3 := 0;
                   #ERR_VAL3 := 0;
                   #ERR_NO4 := 0;
                   #ERR_VAL4 := 0;
                   #ERR_NO5 := 0;
                   #ERR_VAL5 := 0;
                   #ERR_NO6 := 0;
                   #ERR_VAL6 := 0;
                   #ERR_NO7 := 0;
                   #ERR_VAL7 := 0;
                   #ERR_NO8 := 0;
                   #ERR_VAL8 := 0;

                   //Auftrag ist nicht aktiv 

                   #BUSY_AC := FALSE;

                 ELSE
                   //Anzahl Auftragswiederholungen, wenn keine plausiblen Antwortdaten vorhanden, erhoehen 

                   #WDOG_RETRY := #WDOG_RETRY + 1;

                   //Anzahl Zyklen initialisieren 

                   #NODATA_CYCLE := 0;

                   //Auftragswiederholung anstossen 

                   #SEND_AC := TRUE;
                 END_IF;
                 //END_IF of IF #sb_DONE_AC

               END_IF;
               //END_IF of IF #HM_RET_VAL < 0

             END_IF;
             //END_IF of IF #b_busy = FALSE

           ELSE
             ;
             //Watchdog-     
             //Fehler melden 

             #sb_WDOG_ERR := TRUE;

             //Auftrag ist nicht aktiv 

             #BUSY_AC := FALSE;
           END_IF;
           //END_IF of IF #WDOG_RETRY < #WDOG_RETRY_NO

         ELSE
           ;
           //Nein: Keine Bearbeitung 
         END_IF;
         //END_IF of IF #BUSY_AC
       END_IF;
       //END_IF of IF (NOT #BUSY_AC AND #START_AC) OR (#BUSY_AC AND #SEND_AC)
     ELSE
       ;
       //Konfigurationsfehler: Keine weitere Bearbeitung 

       #sb_CFG_ERR := TRUE;

       //Auftrag ist nicht aktiv 

       #BUSY_AC := FALSE;

       //Auftrag fertig ruecksetzen 

       #READY_AC := FALSE;
     END_IF;
     //END_IF of IF (#LADDR <> 16#0000)

     //Stoerungen auslesen: Antwort auswerten 

     //Stoerungen auslesen laeuft 

     IF #sb_BUSY
     THEN
       //Auftrag fertig 

       IF #sb_DONE_AC
       THEN
         //Auftrag fertig ohne Fehler 

         #DONE := TRUE;

         //Auftrag ist nicht aktiv 

         #sb_BUSY := FALSE;
       ELSE
         ;
         //Fehler aufgetreten waehrend der Kommunikation 

         IF #sb_REQ_ERR OR #sb_WDOG_ERR OR #sb_SFB_ERR OR #sb_CFG_ERR
         THEN
           //Auftrag ist nicht aktiv 

           #sb_BUSY := FALSE;

           //Auftrag ist nicht fertig 

           #DONE := FALSE;
         END_IF;
         //END_IF of IF #REQ_ERR OR #WDOG_ERR OR #SFB_ERR OR #CFG_ERR
       END_IF;
       //END_IF of IF #sb_DONE_AC
     END_IF;
     //END_IF of IF #BUSY

     // Initialisierung von Ausg㭧en
     #BUSY := #sb_BUSY;
     #REQ_ERR := #sb_REQ_ERR;
     #WDOG_ERR := #sb_WDOG_ERR;
     #SFB_ERR := #sb_SFB_ERR;
     #CFG_ERR := #sb_CFG_ERR;
END_FUNCTION_BLOCK

// ===== library: MasterCopy "PCD_RECV" =====

FUNCTION_BLOCK "PCD_RECV"   // FB32, STL
TITLE = PCD_RECV
{ S7_Optimized_Access := 'FALSE' }
AUTHOR : DRVDPS7
FAMILY : DRIVES
NAME : PCD_RECV
VERSION : 5.0
// Read process data (CPU 1500)
   VAR_INPUT
      CFG_DATA : "SLOT_UDT";
   END_VAR
   VAR_OUTPUT
      PCD_1 : Word;   // Status word
      PCD_2 : Word;   // Main actual value
      PCD_3 : Word;   // Actual value / Additional status word
      PCD_4 : Word;   // Actual value / Additional status word
      PCD_5 : Word;   // Actual value / Additional status word
      PCD_6 : Word;   // Actual value / Additional status word
      PCD_7 : Word;   // Actual value / Additional status word
      PCD_8 : Word;   // Actual value / Additional status word
      PCD_9 : Word;   // Actual value / Additional status word
      PCD_10 : Word;   // Actual value / Additional status word
      PCD_11 : Word;   // Actual value / Additional status word
      PCD_12 : Word;   // Actual value / Additional status word
      PCD_13 : Word;   // Actual value / Additional status word
      PCD_14 : Word;   // Actual value / Additional status word
      PCD_15 : Word;   // Actual value / Additional status word
      PCD_16 : Word;   // Actual value / Additional status word
      PCD_17 : Word;   // Actual value / Additional status word
      PCD_18 : Word;   // Actual value / Additional status word
      PCD_19 : Word;   // Actual value / Additional status word
      PCD_20 : Word;   // Actual value / Additional status word
      PCD_21 : Word;   // Actual value / Additional status word
      PCD_22 : Word;   // Actual value / Additional status word
      PCD_23 : Word;   // Actual value / Additional status word
      PCD_24 : Word;   // Actual value / Additional status word
      PCD_25 : Word;   // Actual value / Additional status word
      PCD_26 : Word;   // Actual value / Additional status word
      PCD_27 : Word;   // Actual value / Additional status word
      PCD_28 : Word;   // Actual value / Additional status word
      PCD_29 : Word;   // Actual value / Additional status word
      PCD_30 : Word;   // Actual value / Additional status word
      PCD_31 : Word;   // Actual value / Additional status word
      PCD_32 : Word;   // Actual value / Additional status word
      PLC_CTRL : Bool;   // PLC control requested by slave
      DEV_FLT : Bool;   // Drive signals device fault
      DEV_WARNING : Bool;   // Drive signals device warning
      SFC_ERR : Bool;   // SFC signals error
      CFG_ERR : Bool;   // Slave / slot parameterized incorrectly or not at all
   END_VAR
   VAR
      si_SFC_RET_VAL : Int;   // SFC return value
      sy_PCD_ADDR_OLD : Byte;   // Old process data address
      sy_LENGTH_OLD : Byte;   // Old data length
      sb_SFC_ERR : Bool;
      sb_CFG_ERR : Bool;
   END_VAR
   VAR_TEMP
      pa_transfer_data : Any;
      pd_per_addr : DWord;
      pi_ret_val : Int;
      py_length : Byte;
      py_null : Byte;
   END_VAR
BEGIN

REGION Network 1: Konfigurationsdaten prüfen // Netzwerk 1
   // =============================================================================
   // SIEMENS AG
   // (c)Copyright 2017 All Rights Reserved
   // -----------------------------------------------------------------------------
   //  Tested with: S7-1516-3 PN/DP V1.8
   //  Engineering: TIA Portal V14
   //  Restrictions: -
   //  Requirements: S7-1500
   //  Functionality: The block receives process data (status words, actual values) cyclically from the 
   //                 drive in compliance with the relevant consistency conditions.
   // =============================================================================
         SET;
         R     #SFC_ERR;  // SFC-Fehler rücksetzen
         R     #CFG_ERR;  // Konfigurationsfehler rücksetzen
         R     #sb_SFC_ERR;  // SFC-Fehler rücksetzen
         R     #sb_CFG_ERR;  // Konfigurationsfehler rücksetzen

         A(;
         L     B#16#02;
         L     #CFG_DATA.SLOT_ID;  // Slot = Istwert-Slot ?
         <>I;
         );
         A(;
         L     B#16#03;  // oder Slot = kombinierter
         <>I;  // Soll-/Istwert-Slot
         );
         JC    FEHL;  // Nein : Konfigurationsfehler

         L     B#16#00;  // Datenlänge <> 0 oder
         L     #CFG_DATA.LENGTH;
         ==I;
         JC    FEHL;  // Datenlänge + Prozeßdaten-
         L     #CFG_DATA.PCD_ADDR;  // adresse < 32 + 1?
         +I;
         L     B#16#21;
         >I;
         JC    FEHL;  // Nein : Konfigurationsfehler

         L     #CFG_DATA.PCD_ADDR;  // Prozeßdatenadresse <> 0
         L     B#16#00;
         ==I;

   FEHL: S     #sb_CFG_ERR;  // Nein : Konfigurationsfehler
         JCN   NW01;

         L     B#16#00;  //  RET_VAL löschen

         T     #si_SFC_RET_VAL;

   NW01: NOP   0;
END_REGION

REGION Network 2: Änderung der Prozeßdatenadresse / Datenlänge // Netzwerk 2
         L     #sy_PCD_ADDR_OLD;  // Alt-Neu-Vergleich der
         L     #CFG_DATA.PCD_ADDR;  // Prozeßdatenadresse
         T     #sy_PCD_ADDR_OLD;
         <>I;
         JC    LOES;

         L     #sy_LENGTH_OLD;  // Alt-Neu-Vergleich der
         L     #CFG_DATA.LENGTH;  // Datenlänge
         T     #sy_LENGTH_OLD;
         ==I;
         AN    #sb_CFG_ERR;  // Fehler in der Konfiguration
         JC    NW02;

   LOES: L;  // Prozeßdaten ablöschen
         TAR2;
         AD    DW#16#00FF_FFFF;
         +D;
         LAR1;
         L     B#16#08;
   LOP2: T     #py_length;

         L     B#16#00;
         T     D[AR1,P#0.0];
         +AR1  P#4.0;

         L     #py_length;
         LOOP  LOP2;

         A     #sb_CFG_ERR;  // Bei Konfigurationsfehler
         JC    ENDE;  // keine weitere Bearbeitung

   NW02: NOP   0;
END_REGION

REGION Network 3: Datenübertragung mit Direktzugriffen // Netzwerk 3
         L     #CFG_DATA.LENGTH;  // Datenlänge <= 2 Worte
         L     B#16#02;
         >I;  // oder Wortkonsistenz angewählt
         A     #CFG_DATA.CONSIST;  // => Datenübertragung mit
         JC    NW03;  //    Direktzugriffen

         L     B#16#00;  // SFC RET_VAL löschen
         T     #si_SFC_RET_VAL;

         L     #CFG_DATA.LADDR;  // Logische Basisadresse speichern
         SLD   3;
         T     #pd_per_addr;

         L     #CFG_DATA.PCD_ADDR;
         DEC   1;
         SLD   4;
         L;
         +D;
         TAR2;
         AD    DW#16#00FF_FFFF;
         +D;
         LAR1;  // Adresse Prozeßdaten speichern

         L     #CFG_DATA.LENGTH;  // Datenlänge speichern
   LOP3: T     #py_length;  // Länge = 0
         L     B#16#00;
         ==I;
         JC    NW05;  // => Übertragung beendet

         TAK;
         L     B#16#02;  // Länge >= 2 Worte
         <I;
         JC    WORD;

         L     PID[ #pd_per_addr];  // Doppelwort-Befehl
         T     D[AR1,P#0.0];  // Laden der Peripherie

         +AR1  P#4.0;  // Adresse der Prozeßdaten
         L     #pd_per_addr;  // inkrementieren
         L     P#4.0;  // Logische Basisadresse
         +D;  // inkrementieren
         T     #pd_per_addr;

         L     #py_length;  // Länge subtrahieren
         DEC   2;
         JU    LOP3;

   WORD: L     PIW[ #pd_per_addr];  // Wort-Befehl
         T     W[AR1,P#0.0];  // Laden der Peripherie

         +AR1  P#2.0;  // Adresse der Prozeßdaten
         L     #pd_per_addr;  // inkrementieren
         L     P#2.0;  // Logische Basisadresse
         +D;  // inkrementieren
         T     #pd_per_addr;

         L     #py_length;  // Länge subtrahieren
         DEC   1;
         JU    LOP3;

   NW03: NOP   0;
END_REGION

REGION Network 4: Datenübertragung mit SFC DPRD_DAT // Netzwerk 4
         L;  // Zeiger für Datentransfer
         LAR1;  // bilden
         L     W#16#1002;
         T     LW[AR1,P#0.0];
         L     #CFG_DATA.LENGTH;
         SLW   1;
         T     LW[AR1,P#2.0];
         L     DINO;
         T     LW[AR1,P#4.0];
         L     #CFG_DATA.PCD_ADDR;
         DEC   1;
         SLD   4;
         L;
         +D;
         TAR2;
         AD    DW#16#00FF_FFFF;
         +D;
         T     LD[AR1,P#6.0];

         CALL  DPRD_DAT
         ( LADDR   := #CFG_DATA.LADDR,
           RET_VAL := #si_SFC_RET_VAL,
           RECORD  := #pa_transfer_data
         );


         L     #si_SFC_RET_VAL;  // RET_VAL des SFC DPWR_DAT < 0
         L     B#16#00;
         <I;
         =     #sb_SFC_ERR;  // => SFC-Fehler
         JCN   NW05;

         L     B#16#00;
         T     #py_null;

   // Empfangsfach löschen
         CALL  FILL
         ( BVAL    := #py_null,
           RET_VAL := #pi_ret_val,
           BLK     := #pa_transfer_data
         );
END_REGION

REGION Network 5: Zustandswort auswerten // Netzwerk 5
   NW05: SET;
         R     #DEV_FLT;  // Gerätestörung rücksetzen
         R     #DEV_WARNING;  // Gerätewarnung rücksetzen
         R     #PLC_CTRL;  // AG-Führung rücksetzung

         L     #CFG_DATA.PCD_ADDR;  // Zustandswort wurde übertragen
         L     B#16#01;  // => Zustandswort auswerten
         <>I;
         O     #sb_SFC_ERR;  // Auswertung, wenn kein
         JC    ENDE;  // SFC-Fehler

         L;
         LAR1;
         L     W[AR1,P#0.0];
         SRW   4;  // Bit 3 in Zustandswort = 1
         JZ    DWAR;
         SET;
         S     #DEV_FLT;  // => Antrieb meldet Gerätestörung

   DWAR: L;
         LAR1;
         L     W[AR1,P#0.0];
         SRW   8;  // Bit 7 in Zustandswort = 1
         JZ    PLCC;
         SET;
         S     #DEV_WARNING;  // => Antrieb meldet Gerätewarnung

   PLCC: L;
         LAR1;
         L     W[AR1,P#0.0];
         SRW   10;  // Bit 9 in Zustandswort = 1
         JZ    ENDE;
         SET;  // => AG-Führung vom Slave
         S     #PLC_CTRL;  // gefordert
END_REGION

REGION Network 6: Bausteinende // Netzwerk 5
   ENDE: A     #sb_SFC_ERR;
         =     #SFC_ERR;
         A     #sb_CFG_ERR;
         =     #CFG_ERR;

         BE;
END_REGION
END_FUNCTION_BLOCK

// ===== library: MasterCopy "PCD_SEND" =====

FUNCTION_BLOCK "PCD_SEND"   // FB31, STL
TITLE = PCD_SEND
{ S7_Optimized_Access := 'FALSE' }
AUTHOR : DRVDPS7
FAMILY : DRIVES
NAME : PCD_SEND
VERSION : 5.0
// Write process data (CPU 1500)
   VAR_INPUT
      CFG_DATA : "SLOT_UDT";
      PCD_1 : Word;   // Control word
      PCD_2 : Word;   // Main setpoint
      PCD_3 : Word;   // Setpoint / Additional control word
      PCD_4 : Word;   // Setpoint / Additional control word
      PCD_5 : Word;   // Setpoint / Additional control word
      PCD_6 : Word;   // Setpoint / Additional control word
      PCD_7 : Word;   // Setpoint / Additional control word
      PCD_8 : Word;   // Setpoint / Additional control word
      PCD_9 : Word;   // Setpoint / Additional control word
      PCD_10 : Word;   // Setpoint / Additional control word
      PCD_11 : Word;   // Setpoint / Additional control word
      PCD_12 : Word;   // Setpoint / Additional control word
      PCD_13 : Word;   // Setpoint / Additional control word
      PCD_14 : Word;   // Setpoint / Additional control word
      PCD_15 : Word;   // Setpoint / Additional control word
      PCD_16 : Word;   // Setpoint / Additional control word
      PCD_17 : Word;   // Setpoint / Additional control word
      PCD_18 : Word;   // Setpoint / Additional control word
      PCD_19 : Word;   // Setpoint / Additional control word
      PCD_20 : Word;   // Setpoint / Additional control word
      PCD_21 : Word;   // Setpoint / Additional control word
      PCD_22 : Word;   // Setpoint / Additional control word
      PCD_23 : Word;   // Setpoint / Additional control word
      PCD_24 : Word;   // Setpoint / Additional control word
      PCD_25 : Word;   // Setpoint / Additional control word
      PCD_26 : Word;   // Setpoint / Additional control word
      PCD_27 : Word;   // Setpoint / Additional control word
      PCD_28 : Word;   // Setpoint / Additional control word
      PCD_29 : Word;   // Setpoint / Additional control word
      PCD_30 : Word;   // Setpoint / Additional control word
      PCD_31 : Word;   // Setpoint / Additional control word
      PCD_32 : Word;   // Setpoint / Additional control word
   END_VAR
   VAR_OUTPUT
      SFC_ERR : Bool;   // SFC signals error
      CFG_ERR : Bool;   // Slave / slot parameterized incorrectly or not at all
   END_VAR
   VAR
      si_SFC_RET_VAL : Int;   // SFC return value
   END_VAR
   VAR_TEMP
      pa_transfer_data : Any;
      pd_per_addr : DWord;
      py_length : Byte;
   END_VAR
BEGIN

REGION Network 1: Konfigurationsdaten prüfen // Netzwerk 1
   // =============================================================================
   // SIEMENS AG
   // (c)Copyright 2017 All Rights Reserved
   // -----------------------------------------------------------------------------
   //  Library: DriveLib
   //  Tested with: S7-1516-3 PN/DP V1.8
   //  Engineering: TIA Portal V14
   //  Restrictions: -
   //  Requirements: S7-1500
   //  Functionality: Adhering to the relevant consistency conditions, the block transfers the process 
   //                 data (control words, setpoints) cyclically from the SIMATIC to the drive.
   // =============================================================================
         SET;
         R     #SFC_ERR;  // SFC-Fehler rücksetzen
         R     #CFG_ERR;  // Konfigurationsfehler rücksetzen

         A(;
         L     B#16#01;
         L     #CFG_DATA.SLOT_ID;  // Slot = Sollwert-Slot ?
         <>I;
         );
         A(;
         L     B#16#03;  // oder Slot = kombinierter
         <>I;  // Soll-/Istwert-Slot
         );
         JC    FEHL;  // Nein : Konfigurationsfehler

         L     B#16#00;  // Datenlänge <> 0 oder
         L     #CFG_DATA.LENGTH;
         ==I;
         JC    FEHL;  // Datenlänge + Prozeßdaten-
         L     #CFG_DATA.PCD_ADDR;  // adresse < 32 + 1?
         +I;
         L     B#16#21;
         >I;
         JC    FEHL;  // Nein : Konfigurationsfehler

         L     #CFG_DATA.PCD_ADDR;  // Prozeßdatenadresse <> 0
         L     B#16#00;
         ==I;

   FEHL: S     #CFG_ERR;  // Nein : Konfigurationsfehler
         JCN   NW01;

         L     B#16#00;  // SFC RET_VAL löschen
         T     #si_SFC_RET_VAL;
         JU    ENDE;

   NW01: NOP   0;
END_REGION

REGION Network 2: Datenübertragung mit Direktzugriffen // Netzwerk 2
         L     #CFG_DATA.LENGTH;  // Datenlänge <= 2 Worte
         L     B#16#02;
         >I;  // oder Wortkonsistenz angewählt
         A     #CFG_DATA.CONSIST;  // => Datenübertra-gung mit
         JC    NW02;  //    Direktzugriffen

         L     B#16#00;  // SFC RET_VAL löschen
         T     #si_SFC_RET_VAL;

         L     #CFG_DATA.LADDR;  // Logische Basisadresse speichern
         SLD   3;
         T     #pd_per_addr;

         L     #CFG_DATA.PCD_ADDR;
         DEC   1;
         SLD   4;
         L;
         +D;
         TAR2;
         AD    DW#16#00FF_FFFF;
         +D;
         LAR1;  // Adresse Prozeßdaten speichern

         L     #CFG_DATA.LENGTH;  // Datenlänge speichern
   LOP2: T     #py_length;  // Länge = 0
         L     B#16#00;
         ==I;
         JC    ENDE;  // => Übertragung beendet

         TAK;
         L     B#16#02;  // Länge >= 2 Worte
         <I;
         JC    WORD;

         L     D[AR1,P#0.0];  // Doppelwort-Befehl
         T     PQD[ #pd_per_addr];  // Schreiben auf die Peripherie

         +AR1  P#4.0;  // Adresse der Prozeßdaten
         L     #pd_per_addr;  // inkrementieren
         L     P#4.0;  // Logische Basisadresse
         +D;  // inkrementieren
         T     #pd_per_addr;

         L     #py_length;  // Länge subtrahieren
         DEC   2;
         JU    LOP2;

   WORD: L     W[AR1,P#0.0];  // Wort-Befehl
         T     PQW[ #pd_per_addr];  // Schreiben auf die Peripherie

         +AR1  P#2.0;  // Adresse der Prozeßdaten
         L     #pd_per_addr;  // inkrementieren
         L     P#2.0;  // Logische Basisadresse
         +D;  // inkrementieren
         T     #pd_per_addr;

         L     #py_length;  // Länge subtrahieren
         DEC   1;
         JU    LOP2;

   NW02: NOP   0;
END_REGION

REGION Network 3: Datenübertragung mit SFC DPWR_DAT // Netzwerk 3
         L;  // Zeiger für Datentransfer
         LAR1;  // bilden
         L     W#16#1002;
         T     LW[AR1,P#0.0];
         L     #CFG_DATA.LENGTH;
         SLW   1;
         T     LW[AR1,P#2.0];
         L     DINO;
         T     LW[AR1,P#4.0];
         L     #CFG_DATA.PCD_ADDR;
         DEC   1;
         SLD   4;
         L;
         +D;
         TAR2;
         AD    DW#16#00FF_FFFF;
         +D;
         T     LD[AR1,P#6.0];

         CALL  DPWR_DAT
         ( LADDR   := #CFG_DATA.LADDR,
           RECORD  := #pa_transfer_data,
           RET_VAL := #si_SFC_RET_VAL
         );


         L     #si_SFC_RET_VAL;  // RET_VAL des SFC DPWR_DAT < 0
         L     B#16#00;
         <I;
         =     #SFC_ERR;  // => SFC-Fehler
END_REGION

REGION Network 4: Bausteinende // Netzwerk 4
   ENDE: BE;
END_REGION
END_FUNCTION_BLOCK

// ===== library: MasterCopy "PDAT_AC2" =====

FUNCTION_BLOCK "PDAT_AC2"   // FB36, SCL
TITLE = PDAT_AC2
{ S7_Optimized_Access := 'FALSE' }
AUTHOR : DRVDPS7
FAMILY : DRIVES
NAME : PDAT_AC2
VERSION : 5.0
// Process parameters acyclically (CPU 1500)
   VAR_INPUT
      LADDR : HW_IO;   // Logic base address of slot
      START : Bool;   // Accept start impulse for request
      DS_NO : Word := 0;   // Number of data record
      DB_NO_OR : DInt;   // DB No. of order DB
      OFFSET_OR : Int;   // Startaddress of user data in order DB
      DB_NO_AN : DInt;   // DB No. of answer DB
      OFFSET_AN : Int;   // Startaddress of user data in answer DB
   END_VAR
   VAR_OUTPUT
      BUSY : Bool;   // Request busy
      DONE : Bool := 1;   // Request completed without error
      REQ_ERR : Bool;   // Request completed with error
      WDOG_ERR : Bool;   // Watchdog error, no plausible response data exist
      SFB_ERR : Bool;   // SFB 53 WRREC / SFC 52 RDREC signals error
      CFG_ERR : Bool;   // Slave incorrectly configured or not at all
      DB_ERR : Bool;   // Wrong construction of order and/or answer DB
      DB_ERRNO : Int;   // Errorcode to explain DB_ERR
      DB_ACT : DInt;   // DB No. of active order
      OFFSET_ACT : Int;   // Offset of active order
   END_VAR
   VAR
      sb_SEND : Bool;   // Transmission active or request repetition
      sb_START_OLD : Bool := 0;   // Start flag
      sb_CFG_ERR_1 : Bool;   // Fehler bei LADDR
      sb_DB_ERR : Bool;   // Fehler im Auftragsfach
      sb_BUSY : Bool;   // Request busy
      sb_DONE : Bool;   // Request completed without error
      sb_REQ_ERR : Bool;   // Request completed with error
      si_SFB53_RET_VAL : Int;   // Return value of SFB 53 RDREC
      si_SFB52_RET_VAL : Int;   // Return value of SFB 52 WRREC
      si_WDOG_RETRY : Int;   // Counter for request retry for Watchdog monitoring
      si_NODATA_RETRY : Int;   // Counter for request retry if none Response data exist
      si_NODATA_CYCLE : Int;   // Cycle counter, if no reponse data exists
      si_WDOG_RETRY_NO : Int := 5;   // Number of request retries, when no plausible response data exists
      si_NODATA_RETRY_NO : Int := 5;   // Number of request retries, when no response data exist
      si_NODATA_CYCLE_NO : Int := 2500;   // Number of cycles when no response data exist, before request retry
      si_HM_RET_VAL : Int;   // Return value of SFC
      sa_SEND_BUF : Array[0..239] of Byte;   // Send buffer
      sa_RECV_BUF : Array[0..239] of Byte;   // Receive buffer
      WRREC_1 : WRREC;   // Multiinstance of WRREC (SFB53)
      RDREC_1 : RDREC;   // Multiinstance of RDREC (SFB52)
      sb_ATTRIB : Byte;
      sul_DB_LENGTH : UDInt;
      si_ACT_LENGTH : Int;
   END_VAR
   VAR_TEMP
      pb_BUSY : Bool;   // SFB53 / SFB52 aktive
      pb_DONE_WRREC : Bool;   // WRREC fertig
      pb_DONE_RDREC : Bool;   // RDREC fertig
      pb_ERR_WRREC : Bool;   // WRREC Fehler
      pb_ERR_RDREC : Bool;   // RDREC Fehler
      pi_INDEX : Int;   // Index zum Umkopieren der Daten aus dem Sende- / Empfangspuffer aus / in den Auftrags- / Antwort-DB
      pi_LEN_RDREC : UInt;   // Tatsaechliche Laenge der empfangenen Daten
      pi_SFB_INDEX : Int;   // Index bei SFB52/53 Aufruf
      pd_STATUS : DWord;   // STATUS der SFB's
      pl_OFFSET : DInt;
      pi_RET_VAL : Int;
   END_VAR
BEGIN
     //=============================================================================
     //SIEMENS AG
     //(c)Copyright 2017 All Rights Reserved
     //-----------------------------------------------------------------------------
     // Library: DriveLib
     // Tested with: S7-1516-3 PN/DP V1.8
     // Engineering: TIA Portal V14
     // Restrictions: -
     // Requirements: S7-1500
     // Functionality: The block coordinates acyclic communications between the driver and the S7-CPU 
     //                for the transmission of parameter data in accordance with the extended 
     //                PROFIdrive Profile Drive Technology. Data exchange takes place via the S7 
     //                communications services "Read/write data record" (data record number 47). 
     //=============================================================================

     //Konfigurationsdaten pruefen: Logische Basisadresse <> 0 

     IF #LADDR <> 16#0000
     THEN
       //Konfiguration ok 

       #sb_CFG_ERR_1 := FALSE;

       IF #sb_BUSY
       THEN
         IF #si_NODATA_CYCLE < #si_NODATA_CYCLE_NO
         THEN
           //Anzahl Zyklen erhoehen 

           #si_NODATA_CYCLE := #si_NODATA_CYCLE + 1;
         ELSE
           ;
           IF #si_HM_RET_VAL < 0
           THEN
             //Keine Antwortdaten vorhanden? 

             IF #si_NODATA_RETRY < #si_NODATA_RETRY_NO
             THEN
               //Anzahl Auftragswiederholungen erhoehen 

               #si_NODATA_RETRY := #si_NODATA_RETRY + 1;

               //Anzahl Zyklen initialisieren 

               #si_NODATA_CYCLE := 0;
             ELSE
               ;
               //SFC - Fehler 

               #SFB_ERR := TRUE;

               IF #sb_SEND
               THEN
                 //Datensatz schreiben: Keine Antwortdaten vorhanden oder temporaerer Fehler, RET_VAL uebergeben 

                 #si_SFB53_RET_VAL := #si_HM_RET_VAL;
               ELSE
                 ;
                 //Datensatz lesen: Keine Antwortdaten vorhanden oder temporaerer Fehler, RET_VAL uebergeben 

                 #si_SFB52_RET_VAL := #si_HM_RET_VAL;
               END_IF;

               //END_IF of IF #sb_SEND 

               //Auftragswiederholung ruecksetzen 

               #sb_SEND := FALSE;

               //Aufrag nicht aktiv 

               #sb_BUSY := FALSE;
             END_IF;

             //END_IF of IF #si_NODATA_RETRY < #si_NODATA_RETRY 
           ELSE
             ;
             //keine Bedeutung 
           END_IF;

           //END_IF of IF #si_HM_RET_VAL < 0 
         END_IF;

         //END_IF of IF #si_NODATA_CYCLE < #si_NODATA_CYCLE_NO 
       ELSE
         ;
         //Anzahl Zyklen und Anzahl Auftragswiederholungen initialisieren 

         #si_NODATA_CYCLE := 0;
         #si_NODATA_RETRY := 0;
         #si_WDOG_RETRY := 0;
       END_IF;

       //END_IF of IF #BUSY 

       //Ueberpruefung, welcher Datensatz verwendet werden soll 

       #pi_SFB_INDEX := WORD_TO_INT(#DS_NO);

       IF #pi_SFB_INDEX = 0
       THEN
         #pi_SFB_INDEX := 47;
       ELSE
         ;
         ;    // not used
       END_IF;

       IF (NOT #sb_BUSY AND #START AND NOT #sb_START_OLD) OR (#sb_BUSY AND #sb_SEND)
       THEN
         //Senden 

         IF #START AND NOT #sb_START_OLD AND NOT #sb_SEND
         THEN
           //Fehler / Ausgaenge / Hilfsmerker ruecksetzen 

           #sb_DONE := FALSE;
           #sb_REQ_ERR := FALSE;
           #WDOG_ERR := FALSE;
           #SFB_ERR := FALSE;
           #DB_ERR := FALSE;
           #DB_ERRNO := 0;
           #sb_DB_ERR := FALSE;
           #si_SFB53_RET_VAL := 0;
           #si_SFB52_RET_VAL := 0;

           //Auftrags-DB und Offset an die Ausgaenge schreiben 

           #DB_ACT := #DB_NO_OR;
           #OFFSET_ACT := #OFFSET_OR;


           //Auftrags-DB auf Gueltigkeit ueberpruefen 
           #pi_RET_VAL := ATTR_DB(REQ := 1, DB_NUMBER := DINT_TO_UINT(#DB_NO_OR), DB_LENGTH => #sul_DB_LENGTH, ATTRIB => #sb_ATTRIB);

           #si_ACT_LENGTH := #OFFSET_OR + 240;

           IF (#pi_RET_VAL <> 0) OR (UDINT_TO_INT(#sul_DB_LENGTH) < #si_ACT_LENGTH)
           THEN
             #sb_DB_ERR := TRUE;
             #DB_ERRNO := 1;
           END_IF;
           //END_IF of (pi_RET_VAL <> 0) OR (pw_DB_LENGTH_1 >= pw_ACT_LENGTH) 

           //Antwort-DB auf Gueltigkeit ueberpruefen 
           #pi_RET_VAL := ATTR_DB(REQ := 1, DB_NUMBER := DINT_TO_UINT(#DB_NO_AN), DB_LENGTH => #sul_DB_LENGTH, ATTRIB => #sb_ATTRIB);

           #si_ACT_LENGTH := #OFFSET_AN + 240;

           IF (#pi_RET_VAL <> 0) OR (UDINT_TO_INT(#sul_DB_LENGTH) < #si_ACT_LENGTH)
           THEN
             #sb_DB_ERR := TRUE;

             #DB_ERRNO := 2;
           END_IF;
           //END_IF of (pi_RET_VAL <> 0) OR (pw_DB_LENGTH_2 >= pw_ACT_LENGTH) 

           IF NOT #sb_DB_ERR
           THEN
             //Daten aus DB in Sendepuffer kopieren 
             FOR #pi_INDEX := 0 TO 239
             DO
               #pl_OFFSET := INT_TO_DINT(#OFFSET_OR + #pi_INDEX);
               #sa_SEND_BUF[#pi_INDEX] := PEEK(area := 16#84, dbNumber := #DB_NO_OR, byteOffset := #pl_OFFSET);

             END_FOR;
             //END_FOR OF FOR #pi_INDEX := 0 TO 239 

             IF (#sa_SEND_BUF[3] < 1) OR (#sa_SEND_BUF[3] > 39)
             THEN
               #sb_DB_ERR := TRUE;

               #DB_ERRNO := 3;
             ELSE
               ;
               FOR #pi_INDEX := 0 TO (BYTE_TO_INT(#sa_SEND_BUF[3]) - 1)
               DO
                 IF (BYTE_TO_INT(#sa_SEND_BUF[5 + (#pi_INDEX * 6)]) < 0) OR (BYTE_TO_INT(#sa_SEND_BUF[5 + (#pi_INDEX * 6)]) > 234)
                 THEN
                   #sb_DB_ERR := TRUE;

                   #DB_ERRNO := 4;
                 ELSE
                   ;
                   //keine Bedeutung 
                 END_IF;

                 //END_IF of IF (sa_SEND_BUF[5+(pi_INDEX * 6)] < 0) OR sa_SEND_BUF[5+(pi_INDEX * 6)] > 234) 
               END_FOR;

               //END_FOR of FOR #pi_INDEX := 0 TO (BYTE_TO_INT (#sa_SEND_BUF[3])-1)
             END_IF;

             //(#sa_SEND_BUF[3] < 1) OR (#sa_SEND_BUF[3] > 39 ) 
           ELSE
             ;
             //keine Bedeutung 
           END_IF;

           //END_IF of IF NOT #sb_DB_ERR 
         ELSE
           ;
           //keine Bedeutung 
         END_IF;

         //END_IF of IF  #START AND NOT #sb_START_OLD AND NOT #sb_SEND 

         IF NOT #sb_DB_ERR
         THEN
           //Datenuebertragung: Auftrag senden (SFB53) 

           #WRREC_1(REQ := TRUE,
                    ID := #LADDR,
                    INDEX := #pi_SFB_INDEX,
                    LEN := 240,
                    RECORD := #sa_SEND_BUF);
           #pb_DONE_WRREC := #WRREC_1.DONE;
           #pb_BUSY := #WRREC_1.BUSY;
           #pb_ERR_WRREC := #WRREC_1.ERROR;
           #pd_STATUS := #WRREC_1.STATUS AND 16#FFFF00;
           #pd_STATUS := SHR(IN := #pd_STATUS, N := 8);

           #si_HM_RET_VAL := DWORD_TO_INT(#pd_STATUS);

           IF NOT #pb_BUSY
           THEN
             IF #si_HM_RET_VAL < 0
             THEN
               //Temporaerer Fehler: RET_VAL <> 80A7, 80B5, 80C0, 80C1, 80C2, 80C3 oder 80C4 

               IF (#si_HM_RET_VAL <> -32601) AND (#si_HM_RET_VAL <> -32587) AND ((#si_HM_RET_VAL < -32576) OR (#si_HM_RET_VAL > -32572))
               THEN
                 //SFC-Fehler 

                 #SFB_ERR := TRUE;

                 //RET_VAL speichern 

                 #si_SFB53_RET_VAL := #si_HM_RET_VAL;

                 //Senden aktiv / Auftragswiederholung ruecksetzen 

                 #sb_SEND := FALSE;

                 //Auftrag ist nicht aktiv 

                 #sb_BUSY := FALSE;
               ELSE
                 ;
                 //Auftrag ist aktiv 

                 #sb_BUSY := TRUE;

                 //Senden aktiv setzen, Auftrag wird noch einmal geschrieben. 

                 #sb_SEND := TRUE;
               END_IF;

               //END_IF of IF (#si_HM_RET_VAL <> -32601) AND (#si_HM_RET_VAL <> -32587) AND ((#si_HM_RET_VAL < -32576) OR (#si_HM_RET_VAL > -32572))
             ELSE
               ;
               //Auftrag ist aktiv 

               #sb_BUSY := TRUE;

               //Auftragswiederholung ruecksetzen 

               #sb_SEND := FALSE;
             END_IF;

             //END_IF of IF #si_HM_RET_VAL < 0 
           ELSE
             ;
             //Empfangspuffer abloeschen 
             FILL_BLK(IN := b#16#0,
                      COUNT := 240,
                      OUT => #sa_RECV_BUF[0]);


             //Auftrag ist aktiv 

             #sb_BUSY := TRUE;

             //Senden aktiv setzen 

             #sb_SEND := TRUE;
           END_IF;
           //END_IF of IF #pb_BUSY 

         ELSE
           ;
           #sb_BUSY := FALSE;
           #sb_DONE := FALSE;
           #sb_SEND := FALSE;
         END_IF;
         //END_IF of IF NOT sb_DB_ERR

       ELSE
         ;
         //Empfangen 

         IF #sb_BUSY
         THEN
           IF #si_WDOG_RETRY < #si_WDOG_RETRY_NO
           THEN
             //Datenuebertragung: Auftrag empfangen 

             #RDREC_1(REQ := TRUE,
                      ID := #LADDR,
                      INDEX := #pi_SFB_INDEX,
                      MLEN := 240,
                      RECORD := #sa_RECV_BUF);

             #pb_DONE_RDREC := #RDREC_1.VALID;
             #pb_BUSY := #RDREC_1.BUSY;
             #pb_ERR_RDREC := #RDREC_1.ERROR;
             #pd_STATUS := #RDREC_1.STATUS AND 16#FFFF00;
             #pi_LEN_RDREC := #RDREC_1.LEN;

             #pd_STATUS := SHR(IN := #pd_STATUS, N := 8);
             #si_HM_RET_VAL := DWORD_TO_INT(#pd_STATUS);

             IF NOT #pb_BUSY
             THEN
               //SFB-Fehler vorhanden? 

               IF #si_HM_RET_VAL < 0
               THEN
                 //Temporaerer Fehler: RET_VAL <> 80A7, 80B5, 80C0, 80C1, 80C2, 80C3 oder 80C4 

                 IF (#si_HM_RET_VAL <> -32601) AND (#si_HM_RET_VAL <> -32587) AND ((#si_HM_RET_VAL < -32576) OR (#si_HM_RET_VAL > -32572))
                 THEN
                   //SFC-Fehler 

                   #SFB_ERR := TRUE;

                   //RET_VAL speichern 

                   #si_SFB52_RET_VAL := #si_HM_RET_VAL;

                   //Auftrag ist nicht aktiv 

                   #sb_BUSY := FALSE;

                   //Antwortbereich abloeschen 

                   FOR #pi_INDEX := 0 TO 239
                   DO
                     #pl_OFFSET := INT_TO_DINT(#OFFSET_AN + #pi_INDEX);
                     POKE(area := 16#84,
                          dbNumber := #DB_NO_AN,
                          byteOffset := #pl_OFFSET,
                          value := B#16#0);

                   END_FOR;
                   //END_FOR OF FOR #pi_INDEX := 0 TO 239 

                 ELSE
                   ;
                   //keine Bedeutung 
                 END_IF;
                 //END_IF of IF (#si_HM_RET_VAL <> -32601) AND (#si_HM_RET_VAL <> -32587) AND ((#si_HM_RET_VAL < -32576) OR (#si_HM_RET_VAL > -32572))

               ELSE
                 ;
                 //Antwortdaten auswerten 

                 IF #sa_SEND_BUF[0] = #sa_RECV_BUF[0]
                 THEN
                   IF #sa_RECV_BUF[1] = 16#81 OR #sa_RECV_BUF[1] = 16#82
                   THEN
                     #sb_REQ_ERR := TRUE;

                     #sb_DONE := FALSE;
                   ELSE
                     ;
                     #sb_REQ_ERR := FALSE;

                     #sb_DONE := TRUE;
                   END_IF;

                   //END_IF of IF #sa_RECV_BUF[1] = 16#81 OR #sa_RECV_BUF[1] = 16#82
                 ELSE
                   ;
                   //keine Bedeutung 
                 END_IF;

                 //END_IF of IF #sa_SEND_BUF[0] = #sa_RECV_BUF[0]

                 //Auftrag fertig ohne / mit Fehler 

                 IF #sb_DONE OR #sb_REQ_ERR
                 THEN
                   //Antwortdaten  ausgeben 

                   FOR #pi_INDEX := 0 TO 239
                   DO
                     #pl_OFFSET := INT_TO_DINT(#OFFSET_AN + #pi_INDEX);

                     POKE(area := 16#84,
                          dbNumber := #DB_NO_AN,
                          byteOffset := #pl_OFFSET,
                          value := #sa_RECV_BUF[#pi_INDEX]);

                   END_FOR;
                   //END_FOR OF FOR #pi_INDEX := 0 TO 239 

                   //Auftrag nicht aktiv 

                   #sb_BUSY := FALSE;
                 ELSE
                   ;
                   //Anzahl Auftragswiederholungen, wenn keine plausiblen Antwortdaten vorhanden, erhoehen 

                   #si_WDOG_RETRY := #si_WDOG_RETRY + 1;

                   //Anzahl Zyklen initialisieren 

                   #si_NODATA_CYCLE := 0;

                   //Auftragswiederholung anstossen 

                   #sb_SEND := TRUE;
                 END_IF;
                 //END_IF of IF #DONE OR #REQ_ERR

               END_IF;
               //END_IF OF IF #si_HM_RET_VAL < 0

             ELSE
               ;
               //keine Bedeutung 
             END_IF;
             //END_IF of IF NOT #pb_BUSY

           ELSE
             ;
             //Watchdog-Fehler melden 

             #WDOG_ERR := TRUE;

             //Auftrag ist nicht aktiv 

             #sb_BUSY := FALSE;

             //Antwortdaten  ausgeben 

             FOR #pi_INDEX := 0 TO 239
             DO
               #pl_OFFSET := INT_TO_DINT(#OFFSET_AN + #pi_INDEX);

               POKE(area := 16#84,
                    dbNumber := #DB_NO_AN,
                    byteOffset := #pl_OFFSET,
                    value := #sa_RECV_BUF[#pi_INDEX]);

             END_FOR;
             //END_FOR OF FOR #pi_INDEX := 0 TO 239

           END_IF;
           //END_IF of IF #si_WDOG_RETRY < #si_WDOG_RETRY_NO 

         ELSE
           ;
           //keine Bedeutung 
         END_IF;
         //END_IF of IF #BUSY 

       END_IF;
       //END_IF of IF (NOT #BUSY AND #START AND NOT #sb_START_OLD) OR (#BUSY AND #sb_SEND)

     ELSE
       ;
       //Konfigurationsfehler: keine weitere Bearbeitung 

       #sb_CFG_ERR_1 := TRUE;

       //Auftrag ist nicht aktiv 

       #sb_BUSY := FALSE;

       //Auftrag fertig ruecksetzen 

       #sb_DONE := FALSE;
     END_IF;
     //END_IF of IF #LADDR <> 16#0000 

     //Flankenauswertung Startimpuls 

     #sb_START_OLD := #START;

     //CFG_ERR ausgeben 

     #CFG_ERR := #sb_CFG_ERR_1;

     //DB_ERR ausgeben 

     #DB_ERR := #sb_DB_ERR;

     // Initialisierung von Ausg㭧en
     #BUSY := #sb_BUSY;
     #DONE := #sb_DONE;
     #REQ_ERR := #sb_REQ_ERR;
END_FUNCTION_BLOCK

// ===== library: MasterCopy "SINA_INFEED" =====

FUNCTION_BLOCK "SINA_INFEED"   // FB288, SCL
TITLE = 'operate a line module'
{ S7_Optimized_Access := 'TRUE' }
AUTHOR : DRVDPS7
FAMILY : DRIVES
NAME : SINA_INFEED
VERSION : 5.1
// Control basic infeed
   VAR_INPUT
      EnablePrecharging : Bool;   // 0-->1 = Setup the DC Link (BLM/SLM/ALM) (OFF1 = 0-->1) / 0-->1 = Zuschaltung der Vorladung des Zwischenkreises (BLM/SLM/ALM) (OFF1 = 0-->1)
      EnableInfeed : Bool;   // 1 = Enable "active" line modules (only SLM / ALM) / 1 = Aktive Einspeisung einschalten (nur SLM / ALM)
      AckFault : Bool;   // 1 = Acknowledge infeed error / 1 = Fehlerquitierung angestoßen
      ConfigAxis : Word := 16#0003;   // binary programmed input to control all functions in the telegram without its own function block input / Binärcodierter Eingang zur Ansteuerung aller nicht als Bausteineingang verfügbaren Steuerbits
      HWIDSTW : HW_IO;   // Hardware Identifer set point slot / Hardware Identifer des Sollwert Slots
      HWIDZSW : HW_IO;   // Hardware Identifer actual value slot / Hardware Identifer des Istwert Slots
   END_VAR
   VAR_OUTPUT
      Ready : Bool;   // 1 = Infeed ready to power up / 1 = Einspeisung einschaltbereit
      Operation : Bool;   // 1 = Infeed ready for operation / 1 = Einspeisung betriebsbereit
      Run : Bool;   // 1 = Infeed in operation (only SLM / ALM) / 1 = Einspeisung im aktiven Betrieb (nur SLM / ALM)
      Fault : Bool;   // 1 = Infeed error active / 1 = Einspeisung Fehler aktiv
      Lockout : Bool;   // 1 = Infeed lockout active / 1 = Einspeisung Einschaltsperre aktiv
      Warning : Bool;   // 1 = Infeed warning active / 1 = Einspeisung Warnung aktiv
      ZSW1 : Word := 16#0000;   // Infeed Status word / Zustandswort Einspeisung
      Error : Bool;   // Rising edge informs that an error occurred during the execution of / Fehler (FB und Einspeisung)
      Status : Word := 16#7002;   // Status output (7002 = FB in operation; 8xxx = error description - read the manual) / Statusausgabe (7002 = FB in Betrieb; 8xxx = Feherbeschreibung siehe Doku)
      DiagID : Word;   // Error codes of the cyclic system funtion blocks DPWR / DPRD_DAT / Fehlercode der zyklischen Systemfunktionen DPWR / DPRD_DAT
   END_VAR
   VAR
      statStwOnOff : Bool;   // STW 1.0
      statStwOff2 : Bool;   // STW 1.1
      statStwQuickStop : Bool;   // STW 1.2
      statStwOperation : Bool;   // STW 1.3
      statStwReleaseRunup : Bool;   // STW 1.4
      statStwDisMotOp : Bool;   // STW 1.5
      statStwDisRegOp : Bool;   // STW 1.6
      statStwAckFault : Bool;   // STW 1.7
      statStwConductRequested : Bool;   // STW 1.10
      statStwDirectOfRot : Bool;   // STW 1.11
      statSTW1 : Word := 16#0062;
      statReady : Bool;
      statOperation : Bool;
      statRun : Bool;
      statFault : Bool;
      statLockout : Bool;
      statWarning : Bool;
   END_VAR
   VAR_TEMP
      tempRetValDPRD : Int;   // Temporary value for infeed enabled
      tempRetValDPWR : Int;
   END_VAR
   VAR CONSTANT
      STATUS_SUBSEQUENT_CALL : Word := 16#7002;   // Subsequent call of FB
      STATUS_WARN_INFEED : Word := 16#7200;   // Infeed warning active
      STATUS_ERROR_PRE : Word := 16#8400;   // Infeed error with the precharge step
      STATUS_ERROR_INF : Word := 16#8401;   // Infeed error (general)
      STATUS_ERROR_DPRD_DAT : Word := 16#8600;   // Error "Read cyclic data" operation
      STATUS_ERROR_DPWR_DAT : Word := 16#8601;   // Error "Write cyclic data" operation
   END_VAR
BEGIN
   //=============================================================================
   //SIEMENS AG
   //(c)Copyright 2017 All Rights Reserved
   //-----------------------------------------------------------------------------
   // Library: DriveLib
   // Tested with: S7-1516-3 PN/DP V1.8
   // Engineering: TIA Portal V14
   // Restrictions: -
   // Requirements: S7-1200 / S7-1500
   // Functionality: the block serves to supply a rectifier unit line module
   //-----------------------------------------------------------------------------
   // Change log table:
   // Version Date       Expert in charge Changes applied
   // 0.1     28.09.2015 ZP               First released version
   // 0.2     09.11.2015 ZP               no internal acknowledgment
   // 0.3     30.11.2015 ZP               new input parameter ConfigAxis
   // 5.0     11.01.2017 FG               adapt version to new DriveLib version
   // 5.1     02.05.2018 FG               Connect all bits from ConfigAxis with
   //                                     the Bits from STW1
   //=============================================================================

   // presetting STW1
   #statStwOnOff := FALSE;     // STW1.0
   #statStwOperation := FALSE;     // STW1.3
   #statStwAckFault := FALSE;      // STW1.7
   #statStwConductRequested := true; //STW1.10 conduct requested set cyclic

   // external setting of STW1
   #statStwOff2 := #ConfigAxis.%X0;  // TRUE if "ConfigAxis" is not assigned STW1.1

   // #statStwQuickStop := #ConfigAxis.%X1; // STW1.2
   // #statStwReleaseRunup := #ConfigAxis.%X2;  // STW1.4      

   #statStwDisMotOp := #ConfigAxis.%X3;  // TRUE if "ConfigAxis" is not assigned STW1.5
   #statStwDisRegOp := #ConfigAxis.%X4; // TRUE if "ConfigAxis" is not assigned STW1.6

   // #statStwDirectOfRot := #ConfigAxis.%X5;  // STW1.11

   // reset error
   #Error := FALSE;
   // acknowledge fault?

   IF #AckFault THEN
     #statStwAckFault := TRUE;  // input AckFault into STW1.7
   END_IF;

   // read status word
   #tempRetValDPRD := DPRD_DAT(LADDR := #HWIDZSW, RECORD => #ZSW1);

   //==========================================
   //#ZSW1 := "SIM_ZSW1";  // only for test
   //==========================================

   // write status word into static word
   #statReady := #ZSW1.%X0;
   #statOperation := #ZSW1.%X1;
   #statRun := #ZSW1.%X2;
   #statFault := #ZSW1.%X3;
   #statLockout := #ZSW1.%X6;
   #statWarning := #ZSW1.%X7;

   // write status word to output
   #Ready := #statReady;
   #Operation := #statOperation;
   #Run := #statRun;
   #Fault := #statFault;
   #Lockout := #statLockout;
   #Warning := #statWarning;

   // Check preconditions
   IF #EnablePrecharging AND #Ready AND NOT #Lockout AND NOT #Fault THEN
     #statStwOnOff := TRUE;      // STW1.0 
     //  #statStwAckFault := FALSE;      // STW1.7
   END_IF;

   (*
   IF #EnablePrecharging AND (NOT #Ready OR #Lockout) THEN
       #statStwOnOff := FALSE;     // STW1.0 
       #statStwOperation := FALSE;     // STW1.3
   END_IF;
   *)

   (* no internal acknowledgment 
   IF #EnablePrecharging AND #Fault THEN  //AND #Ready AND NOT #Lockout
     #statStwOperation := FALSE;     // STW1.3
     #statStwOnOff := FALSE;     // STW1.0
   END_IF;
   *)

   IF #EnablePrecharging AND #Ready AND NOT #Lockout AND NOT #Fault AND NOT #EnableInfeed THEN
     #statStwOperation := FALSE;     // STW1.3
   END_IF;

   IF #EnablePrecharging AND #Ready AND NOT #Lockout AND NOT #Fault AND #EnableInfeed AND NOT #Operation THEN
     #statStwOperation := FALSE;     // STW1.3
   END_IF;

   IF #EnablePrecharging AND #Ready AND NOT #Lockout AND NOT #Fault AND #EnableInfeed AND #Ready AND #Operation THEN
     #statStwOperation := TRUE;     // STW1.3
   END_IF;

   //Error handling and diagnistic DPRD_DAT / DPWR_DAT 
   #Status := #STATUS_SUBSEQUENT_CALL;     // no error activ 16#7002

   IF (NOT #EnablePrecharging AND #EnableInfeed) THEN
     #Error := TRUE;
     #Status := #STATUS_ERROR_PRE; // error precharching 16#8400
     #statStwOperation := FALSE;     // STW1.3 
     #statStwOnOff := FALSE;     // STW1.0
   END_IF;

   IF (NOT #EnablePrecharging AND NOT #EnableInfeed) THEN
     #statStwOperation := FALSE;     // STW1.3 
     #statStwOnOff := FALSE;     // STW1.0
   END_IF;

   // write control word - internal 
   #statSTW1.%X0 := #statStwOnOff;
   #statSTW1.%X3 := #statStwOperation;
   #statSTW1.%X7 := #statStwAckFault;
   #statSTW1.%X10 := #statStwConductRequested;
   // write control word - external 
   #statSTW1.%X1 := #statStwOff2;
   #statSTW1.%X2 := #ConfigAxis.%X4;
   #statSTW1.%X4 := #ConfigAxis.%X5;
   #statSTW1.%X5 := #statStwDisMotOp;
   #statSTW1.%X6 := #statStwDisRegOp;
   #statSTW1.%X8 := #ConfigAxis.%X6;
   #statSTW1.%X9 := #ConfigAxis.%X7;
   #statSTW1.%X11 := #ConfigAxis.%X8;
   #statSTW1.%X12 := #ConfigAxis.%X9;
   #statSTW1.%X13 := #ConfigAxis.%X10;
   #statSTW1.%X14 := #ConfigAxis.%X11;
   #statSTW1.%X15 := #ConfigAxis.%X12;

   #tempRetValDPWR := DPWR_DAT(LADDR := #HWIDSTW, RECORD := #statSTW1); // write STW1

   //======================================
   //"SIM_STW1" := #statSTW1;  // only for test
   //======================================

   #DiagID := 16#0;

   IF #Warning THEN
     #Status := #STATUS_WARN_INFEED;     // warning infeed 16#7200
   ELSIF #Fault THEN
     #Status := #STATUS_ERROR_INF;       // error infeed 16#8401
   ELSIF #tempRetValDPRD <> 16#0 THEN
     #Status := #STATUS_ERROR_DPRD_DAT;       // error code DPRD_DAT 16#8600
     #DiagID := INT_TO_WORD(#tempRetValDPRD);        // diagnistic DPRD_DAT
     #Error := TRUE;
   ELSIF #tempRetValDPWR <> 16#0 THEN
     #Status := #STATUS_ERROR_DPWR_DAT;       // error code DPWR_DAT 16#8601
     #DiagID := INT_TO_WORD(#tempRetValDPWR);        // diagnistic DPWR_DAT
     #Error := TRUE;
   END_IF;
END_FUNCTION_BLOCK

// ===== library: MasterCopy "SINA_PARA" =====

